// NeuroPLC ¡ª FourierKAN L0-direct configuration [28,16,4]
// L0 (28->16): analytic SIN/COS harmonics + SiLU base (no LUT)
// L1 (16->4): LUT N=16 on [-3.15, 3.15] (100% L0-out coverage)
// Sound bound 0.130 (safety 5.2x) ¡ª verify_fourier_l0direct.py
FUNCTION_BLOCK "NeuroPLC_FourierKAN_L0DIR"
VAR_INPUT
    "feat_1" : REAL;
    "feat_2" : REAL;
    "feat_3" : REAL;
    "feat_4" : REAL;
    "feat_5" : REAL;
    "feat_6" : REAL;
    "feat_7" : REAL;
    "feat_8" : REAL;
    "feat_9" : REAL;
    "feat_10" : REAL;
    "feat_11" : REAL;
    "feat_12" : REAL;
    "feat_13" : REAL;
    "feat_14" : REAL;
    "feat_15" : REAL;
    "feat_16" : REAL;
    "feat_17" : REAL;
    "feat_18" : REAL;
    "feat_19" : REAL;
    "feat_20" : REAL;
    "feat_21" : REAL;
    "feat_22" : REAL;
    "feat_23" : REAL;
    "feat_24" : REAL;
    "feat_25" : REAL;
    "feat_26" : REAL;
    "feat_27" : REAL;
    "feat_28" : REAL;
    "trigger" : BOOL;
END_VAR
VAR_OUTPUT
    "class_1" : REAL;
    "class_2" : REAL;
    "class_3" : REAL;
    "class_4" : REAL;
    "pred_class" : INT;
END_VAR
VAR
    "h1_1" : REAL := 0.0;
    "h1_2" : REAL := 0.0;
    "h1_3" : REAL := 0.0;
    "h1_4" : REAL := 0.0;
    "h1_5" : REAL := 0.0;
    "h1_6" : REAL := 0.0;
    "h1_7" : REAL := 0.0;
    "h1_8" : REAL := 0.0;
    "h1_9" : REAL := 0.0;
    "h1_10" : REAL := 0.0;
    "h1_11" : REAL := 0.0;
    "h1_12" : REAL := 0.0;
    "h1_13" : REAL := 0.0;
    "h1_14" : REAL := 0.0;
    "h1_15" : REAL := 0.0;
    "h1_16" : REAL := 0.0;
    "x" : REAL; "phi" : REAL; "acc" : REAL := 0.0;
    "i" : INT; "j" : INT; "k" : INT;
    "lo" : INT; "hi" : INT; "mid" : INT; "t" : REAL;
END_VAR

BEGIN
    IF NOT "trigger" THEN RETURN; END_IF;

    // === L0 (28->16): analytic FourierKAN ===
    "acc" := 0.0;
    "x" := "feat_1";
    "phi" := "w0b_1_1" * "x" / (1.0 + EXP(-"x"));
    "phi" := "phi" + "w0c_1_1_1" * SIN(1 * 0.4 * "x") + "w0d_1_1_1" * COS(1 * 0.4 * "x");
    "phi" := "phi" + "w0c_1_1_2" * SIN(2 * 0.4 * "x") + "w0d_1_1_2" * COS(2 * 0.4 * "x");
    "phi" := "phi" + "w0c_1_1_3" * SIN(3 * 0.4 * "x") + "w0d_1_1_3" * COS(3 * 0.4 * "x");
    "phi" := "phi" + "w0c_1_1_4" * SIN(4 * 0.4 * "x") + "w0d_1_1_4" * COS(4 * 0.4 * "x");
    "phi" := "phi" + "w0c_1_1_5" * SIN(5 * 0.4 * "x") + "w0d_1_1_5" * COS(5 * 0.4 * "x");
    "phi" := "phi" + "w0c_1_1_6" * SIN(6 * 0.4 * "x") + "w0d_1_1_6" * COS(6 * 0.4 * "x");
    "acc" := "acc" + "phi";
    "x" := "feat_2";
    "phi" := "w0b_1_2" * "x" / (1.0 + EXP(-"x"));
    "phi" := "phi" + "w0c_1_2_1" * SIN(1 * 0.4 * "x") + "w0d_1_2_1" * COS(1 * 0.4 * "x");
    "phi" := "phi" + "w0c_1_2_2" * SIN(2 * 0.4 * "x") + "w0d_1_2_2" * COS(2 * 0.4 * "x");
    "phi" := "phi" + "w0c_1_2_3" * SIN(3 * 0.4 * "x") + "w0d_1_2_3" * COS(3 * 0.4 * "x");
    "phi" := "phi" + "w0c_1_2_4" * SIN(4 * 0.4 * "x") + "w0d_1_2_4" * COS(4 * 0.4 * "x");
    "phi" := "phi" + "w0c_1_2_5" * SIN(5 * 0.4 * "x") + "w0d_1_2_5" * COS(5 * 0.4 * "x");
    "phi" := "phi" + "w0c_1_2_6" * SIN(6 * 0.4 * "x") + "w0d_1_2_6" * COS(6 * 0.4 * "x");
    "acc" := "acc" + "phi";
    "x" := "feat_3";
    "phi" := "w0b_1_3" * "x" / (1.0 + EXP(-"x"));
    "phi" := "phi" + "w0c_1_3_1" * SIN(1 * 0.4 * "x") + "w0d_1_3_1" * COS(1 * 0.4 * "x");
    "phi" := "phi" + "w0c_1_3_2" * SIN(2 * 0.4 * "x") + "w0d_1_3_2" * COS(2 * 0.4 * "x");
    "phi" := "phi" + "w0c_1_3_3" * SIN(3 * 0.4 * "x") + "w0d_1_3_3" * COS(3 * 0.4 * "x");
    "phi" := "phi" + "w0c_1_3_4" * SIN(4 * 0.4 * "x") + "w0d_1_3_4" * COS(4 * 0.4 * "x");
    "phi" := "phi" + "w0c_1_3_5" * SIN(5 * 0.4 * "x") + "w0d_1_3_5" * COS(5 * 0.4 * "x");
    "phi" := "phi" + "w0c_1_3_6" * SIN(6 * 0.4 * "x") + "w0d_1_3_6" * COS(6 * 0.4 * "x");
    "acc" := "acc" + "phi";
    "x" := "feat_4";
    "phi" := "w0b_1_4" * "x" / (1.0 + EXP(-"x"));
    "phi" := "phi" + "w0c_1_4_1" * SIN(1 * 0.4 * "x") + "w0d_1_4_1" * COS(1 * 0.4 * "x");
    "phi" := "phi" + "w0c_1_4_2" * SIN(2 * 0.4 * "x") + "w0d_1_4_2" * COS(2 * 0.4 * "x");
    "phi" := "phi" + "w0c_1_4_3" * SIN(3 * 0.4 * "x") + "w0d_1_4_3" * COS(3 * 0.4 * "x");
    "phi" := "phi" + "w0c_1_4_4" * SIN(4 * 0.4 * "x") + "w0d_1_4_4" * COS(4 * 0.4 * "x");
    "phi" := "phi" + "w0c_1_4_5" * SIN(5 * 0.4 * "x") + "w0d_1_4_5" * COS(5 * 0.4 * "x");
    "phi" := "phi" + "w0c_1_4_6" * SIN(6 * 0.4 * "x") + "w0d_1_4_6" * COS(6 * 0.4 * "x");
    "acc" := "acc" + "phi";
    "x" := "feat_5";
    "phi" := "w0b_1_5" * "x" / (1.0 + EXP(-"x"));
    "phi" := "phi" + "w0c_1_5_1" * SIN(1 * 0.4 * "x") + "w0d_1_5_1" * COS(1 * 0.4 * "x");
    "phi" := "phi" + "w0c_1_5_2" * SIN(2 * 0.4 * "x") + "w0d_1_5_2" * COS(2 * 0.4 * "x");
    "phi" := "phi" + "w0c_1_5_3" * SIN(3 * 0.4 * "x") + "w0d_1_5_3" * COS(3 * 0.4 * "x");
    "phi" := "phi" + "w0c_1_5_4" * SIN(4 * 0.4 * "x") + "w0d_1_5_4" * COS(4 * 0.4 * "x");
    "phi" := "phi" + "w0c_1_5_5" * SIN(5 * 0.4 * "x") + "w0d_1_5_5" * COS(5 * 0.4 * "x");
    "phi" := "phi" + "w0c_1_5_6" * SIN(6 * 0.4 * "x") + "w0d_1_5_6" * COS(6 * 0.4 * "x");
    "acc" := "acc" + "phi";
    "x" := "feat_6";
    "phi" := "w0b_1_6" * "x" / (1.0 + EXP(-"x"));
    "phi" := "phi" + "w0c_1_6_1" * SIN(1 * 0.4 * "x") + "w0d_1_6_1" * COS(1 * 0.4 * "x");
    "phi" := "phi" + "w0c_1_6_2" * SIN(2 * 0.4 * "x") + "w0d_1_6_2" * COS(2 * 0.4 * "x");
    "phi" := "phi" + "w0c_1_6_3" * SIN(3 * 0.4 * "x") + "w0d_1_6_3" * COS(3 * 0.4 * "x");
    "phi" := "phi" + "w0c_1_6_4" * SIN(4 * 0.4 * "x") + "w0d_1_6_4" * COS(4 * 0.4 * "x");
    "phi" := "phi" + "w0c_1_6_5" * SIN(5 * 0.4 * "x") + "w0d_1_6_5" * COS(5 * 0.4 * "x");
    "phi" := "phi" + "w0c_1_6_6" * SIN(6 * 0.4 * "x") + "w0d_1_6_6" * COS(6 * 0.4 * "x");
    "acc" := "acc" + "phi";
    "x" := "feat_7";
    "phi" := "w0b_1_7" * "x" / (1.0 + EXP(-"x"));
    "phi" := "phi" + "w0c_1_7_1" * SIN(1 * 0.4 * "x") + "w0d_1_7_1" * COS(1 * 0.4 * "x");
    "phi" := "phi" + "w0c_1_7_2" * SIN(2 * 0.4 * "x") + "w0d_1_7_2" * COS(2 * 0.4 * "x");
    "phi" := "phi" + "w0c_1_7_3" * SIN(3 * 0.4 * "x") + "w0d_1_7_3" * COS(3 * 0.4 * "x");
    "phi" := "phi" + "w0c_1_7_4" * SIN(4 * 0.4 * "x") + "w0d_1_7_4" * COS(4 * 0.4 * "x");
    "phi" := "phi" + "w0c_1_7_5" * SIN(5 * 0.4 * "x") + "w0d_1_7_5" * COS(5 * 0.4 * "x");
    "phi" := "phi" + "w0c_1_7_6" * SIN(6 * 0.4 * "x") + "w0d_1_7_6" * COS(6 * 0.4 * "x");
    "acc" := "acc" + "phi";
    "x" := "feat_8";
    "phi" := "w0b_1_8" * "x" / (1.0 + EXP(-"x"));
    "phi" := "phi" + "w0c_1_8_1" * SIN(1 * 0.4 * "x") + "w0d_1_8_1" * COS(1 * 0.4 * "x");
    "phi" := "phi" + "w0c_1_8_2" * SIN(2 * 0.4 * "x") + "w0d_1_8_2" * COS(2 * 0.4 * "x");
    "phi" := "phi" + "w0c_1_8_3" * SIN(3 * 0.4 * "x") + "w0d_1_8_3" * COS(3 * 0.4 * "x");
    "phi" := "phi" + "w0c_1_8_4" * SIN(4 * 0.4 * "x") + "w0d_1_8_4" * COS(4 * 0.4 * "x");
    "phi" := "phi" + "w0c_1_8_5" * SIN(5 * 0.4 * "x") + "w0d_1_8_5" * COS(5 * 0.4 * "x");
    "phi" := "phi" + "w0c_1_8_6" * SIN(6 * 0.4 * "x") + "w0d_1_8_6" * COS(6 * 0.4 * "x");
    "acc" := "acc" + "phi";
    "x" := "feat_9";
    "phi" := "w0b_1_9" * "x" / (1.0 + EXP(-"x"));
    "phi" := "phi" + "w0c_1_9_1" * SIN(1 * 0.4 * "x") + "w0d_1_9_1" * COS(1 * 0.4 * "x");
    "phi" := "phi" + "w0c_1_9_2" * SIN(2 * 0.4 * "x") + "w0d_1_9_2" * COS(2 * 0.4 * "x");
    "phi" := "phi" + "w0c_1_9_3" * SIN(3 * 0.4 * "x") + "w0d_1_9_3" * COS(3 * 0.4 * "x");
    "phi" := "phi" + "w0c_1_9_4" * SIN(4 * 0.4 * "x") + "w0d_1_9_4" * COS(4 * 0.4 * "x");
    "phi" := "phi" + "w0c_1_9_5" * SIN(5 * 0.4 * "x") + "w0d_1_9_5" * COS(5 * 0.4 * "x");
    "phi" := "phi" + "w0c_1_9_6" * SIN(6 * 0.4 * "x") + "w0d_1_9_6" * COS(6 * 0.4 * "x");
    "acc" := "acc" + "phi";
    "x" := "feat_10";
    "phi" := "w0b_1_10" * "x" / (1.0 + EXP(-"x"));
    "phi" := "phi" + "w0c_1_10_1" * SIN(1 * 0.4 * "x") + "w0d_1_10_1" * COS(1 * 0.4 * "x");
    "phi" := "phi" + "w0c_1_10_2" * SIN(2 * 0.4 * "x") + "w0d_1_10_2" * COS(2 * 0.4 * "x");
    "phi" := "phi" + "w0c_1_10_3" * SIN(3 * 0.4 * "x") + "w0d_1_10_3" * COS(3 * 0.4 * "x");
    "phi" := "phi" + "w0c_1_10_4" * SIN(4 * 0.4 * "x") + "w0d_1_10_4" * COS(4 * 0.4 * "x");
    "phi" := "phi" + "w0c_1_10_5" * SIN(5 * 0.4 * "x") + "w0d_1_10_5" * COS(5 * 0.4 * "x");
    "phi" := "phi" + "w0c_1_10_6" * SIN(6 * 0.4 * "x") + "w0d_1_10_6" * COS(6 * 0.4 * "x");
    "acc" := "acc" + "phi";
    "x" := "feat_11";
    "phi" := "w0b_1_11" * "x" / (1.0 + EXP(-"x"));
    "phi" := "phi" + "w0c_1_11_1" * SIN(1 * 0.4 * "x") + "w0d_1_11_1" * COS(1 * 0.4 * "x");
    "phi" := "phi" + "w0c_1_11_2" * SIN(2 * 0.4 * "x") + "w0d_1_11_2" * COS(2 * 0.4 * "x");
    "phi" := "phi" + "w0c_1_11_3" * SIN(3 * 0.4 * "x") + "w0d_1_11_3" * COS(3 * 0.4 * "x");
    "phi" := "phi" + "w0c_1_11_4" * SIN(4 * 0.4 * "x") + "w0d_1_11_4" * COS(4 * 0.4 * "x");
    "phi" := "phi" + "w0c_1_11_5" * SIN(5 * 0.4 * "x") + "w0d_1_11_5" * COS(5 * 0.4 * "x");
    "phi" := "phi" + "w0c_1_11_6" * SIN(6 * 0.4 * "x") + "w0d_1_11_6" * COS(6 * 0.4 * "x");
    "acc" := "acc" + "phi";
    "x" := "feat_12";
    "phi" := "w0b_1_12" * "x" / (1.0 + EXP(-"x"));
    "phi" := "phi" + "w0c_1_12_1" * SIN(1 * 0.4 * "x") + "w0d_1_12_1" * COS(1 * 0.4 * "x");
    "phi" := "phi" + "w0c_1_12_2" * SIN(2 * 0.4 * "x") + "w0d_1_12_2" * COS(2 * 0.4 * "x");
    "phi" := "phi" + "w0c_1_12_3" * SIN(3 * 0.4 * "x") + "w0d_1_12_3" * COS(3 * 0.4 * "x");
    "phi" := "phi" + "w0c_1_12_4" * SIN(4 * 0.4 * "x") + "w0d_1_12_4" * COS(4 * 0.4 * "x");
    "phi" := "phi" + "w0c_1_12_5" * SIN(5 * 0.4 * "x") + "w0d_1_12_5" * COS(5 * 0.4 * "x");
    "phi" := "phi" + "w0c_1_12_6" * SIN(6 * 0.4 * "x") + "w0d_1_12_6" * COS(6 * 0.4 * "x");
    "acc" := "acc" + "phi";
    "x" := "feat_13";
    "phi" := "w0b_1_13" * "x" / (1.0 + EXP(-"x"));
    "phi" := "phi" + "w0c_1_13_1" * SIN(1 * 0.4 * "x") + "w0d_1_13_1" * COS(1 * 0.4 * "x");
    "phi" := "phi" + "w0c_1_13_2" * SIN(2 * 0.4 * "x") + "w0d_1_13_2" * COS(2 * 0.4 * "x");
    "phi" := "phi" + "w0c_1_13_3" * SIN(3 * 0.4 * "x") + "w0d_1_13_3" * COS(3 * 0.4 * "x");
    "phi" := "phi" + "w0c_1_13_4" * SIN(4 * 0.4 * "x") + "w0d_1_13_4" * COS(4 * 0.4 * "x");
    "phi" := "phi" + "w0c_1_13_5" * SIN(5 * 0.4 * "x") + "w0d_1_13_5" * COS(5 * 0.4 * "x");
    "phi" := "phi" + "w0c_1_13_6" * SIN(6 * 0.4 * "x") + "w0d_1_13_6" * COS(6 * 0.4 * "x");
    "acc" := "acc" + "phi";
    "x" := "feat_14";
    "phi" := "w0b_1_14" * "x" / (1.0 + EXP(-"x"));
    "phi" := "phi" + "w0c_1_14_1" * SIN(1 * 0.4 * "x") + "w0d_1_14_1" * COS(1 * 0.4 * "x");
    "phi" := "phi" + "w0c_1_14_2" * SIN(2 * 0.4 * "x") + "w0d_1_14_2" * COS(2 * 0.4 * "x");
    "phi" := "phi" + "w0c_1_14_3" * SIN(3 * 0.4 * "x") + "w0d_1_14_3" * COS(3 * 0.4 * "x");
    "phi" := "phi" + "w0c_1_14_4" * SIN(4 * 0.4 * "x") + "w0d_1_14_4" * COS(4 * 0.4 * "x");
    "phi" := "phi" + "w0c_1_14_5" * SIN(5 * 0.4 * "x") + "w0d_1_14_5" * COS(5 * 0.4 * "x");
    "phi" := "phi" + "w0c_1_14_6" * SIN(6 * 0.4 * "x") + "w0d_1_14_6" * COS(6 * 0.4 * "x");
    "acc" := "acc" + "phi";
    "x" := "feat_15";
    "phi" := "w0b_1_15" * "x" / (1.0 + EXP(-"x"));
    "phi" := "phi" + "w0c_1_15_1" * SIN(1 * 0.4 * "x") + "w0d_1_15_1" * COS(1 * 0.4 * "x");
    "phi" := "phi" + "w0c_1_15_2" * SIN(2 * 0.4 * "x") + "w0d_1_15_2" * COS(2 * 0.4 * "x");
    "phi" := "phi" + "w0c_1_15_3" * SIN(3 * 0.4 * "x") + "w0d_1_15_3" * COS(3 * 0.4 * "x");
    "phi" := "phi" + "w0c_1_15_4" * SIN(4 * 0.4 * "x") + "w0d_1_15_4" * COS(4 * 0.4 * "x");
    "phi" := "phi" + "w0c_1_15_5" * SIN(5 * 0.4 * "x") + "w0d_1_15_5" * COS(5 * 0.4 * "x");
    "phi" := "phi" + "w0c_1_15_6" * SIN(6 * 0.4 * "x") + "w0d_1_15_6" * COS(6 * 0.4 * "x");
    "acc" := "acc" + "phi";
    "x" := "feat_16";
    "phi" := "w0b_1_16" * "x" / (1.0 + EXP(-"x"));
    "phi" := "phi" + "w0c_1_16_1" * SIN(1 * 0.4 * "x") + "w0d_1_16_1" * COS(1 * 0.4 * "x");
    "phi" := "phi" + "w0c_1_16_2" * SIN(2 * 0.4 * "x") + "w0d_1_16_2" * COS(2 * 0.4 * "x");
    "phi" := "phi" + "w0c_1_16_3" * SIN(3 * 0.4 * "x") + "w0d_1_16_3" * COS(3 * 0.4 * "x");
    "phi" := "phi" + "w0c_1_16_4" * SIN(4 * 0.4 * "x") + "w0d_1_16_4" * COS(4 * 0.4 * "x");
    "phi" := "phi" + "w0c_1_16_5" * SIN(5 * 0.4 * "x") + "w0d_1_16_5" * COS(5 * 0.4 * "x");
    "phi" := "phi" + "w0c_1_16_6" * SIN(6 * 0.4 * "x") + "w0d_1_16_6" * COS(6 * 0.4 * "x");
    "acc" := "acc" + "phi";
    "x" := "feat_17";
    "phi" := "w0b_1_17" * "x" / (1.0 + EXP(-"x"));
    "phi" := "phi" + "w0c_1_17_1" * SIN(1 * 0.4 * "x") + "w0d_1_17_1" * COS(1 * 0.4 * "x");
    "phi" := "phi" + "w0c_1_17_2" * SIN(2 * 0.4 * "x") + "w0d_1_17_2" * COS(2 * 0.4 * "x");
    "phi" := "phi" + "w0c_1_17_3" * SIN(3 * 0.4 * "x") + "w0d_1_17_3" * COS(3 * 0.4 * "x");
    "phi" := "phi" + "w0c_1_17_4" * SIN(4 * 0.4 * "x") + "w0d_1_17_4" * COS(4 * 0.4 * "x");
    "phi" := "phi" + "w0c_1_17_5" * SIN(5 * 0.4 * "x") + "w0d_1_17_5" * COS(5 * 0.4 * "x");
    "phi" := "phi" + "w0c_1_17_6" * SIN(6 * 0.4 * "x") + "w0d_1_17_6" * COS(6 * 0.4 * "x");
    "acc" := "acc" + "phi";
    "x" := "feat_18";
    "phi" := "w0b_1_18" * "x" / (1.0 + EXP(-"x"));
    "phi" := "phi" + "w0c_1_18_1" * SIN(1 * 0.4 * "x") + "w0d_1_18_1" * COS(1 * 0.4 * "x");
    "phi" := "phi" + "w0c_1_18_2" * SIN(2 * 0.4 * "x") + "w0d_1_18_2" * COS(2 * 0.4 * "x");
    "phi" := "phi" + "w0c_1_18_3" * SIN(3 * 0.4 * "x") + "w0d_1_18_3" * COS(3 * 0.4 * "x");
    "phi" := "phi" + "w0c_1_18_4" * SIN(4 * 0.4 * "x") + "w0d_1_18_4" * COS(4 * 0.4 * "x");
    "phi" := "phi" + "w0c_1_18_5" * SIN(5 * 0.4 * "x") + "w0d_1_18_5" * COS(5 * 0.4 * "x");
    "phi" := "phi" + "w0c_1_18_6" * SIN(6 * 0.4 * "x") + "w0d_1_18_6" * COS(6 * 0.4 * "x");
    "acc" := "acc" + "phi";
    "x" := "feat_19";
    "phi" := "w0b_1_19" * "x" / (1.0 + EXP(-"x"));
    "phi" := "phi" + "w0c_1_19_1" * SIN(1 * 0.4 * "x") + "w0d_1_19_1" * COS(1 * 0.4 * "x");
    "phi" := "phi" + "w0c_1_19_2" * SIN(2 * 0.4 * "x") + "w0d_1_19_2" * COS(2 * 0.4 * "x");
    "phi" := "phi" + "w0c_1_19_3" * SIN(3 * 0.4 * "x") + "w0d_1_19_3" * COS(3 * 0.4 * "x");
    "phi" := "phi" + "w0c_1_19_4" * SIN(4 * 0.4 * "x") + "w0d_1_19_4" * COS(4 * 0.4 * "x");
    "phi" := "phi" + "w0c_1_19_5" * SIN(5 * 0.4 * "x") + "w0d_1_19_5" * COS(5 * 0.4 * "x");
    "phi" := "phi" + "w0c_1_19_6" * SIN(6 * 0.4 * "x") + "w0d_1_19_6" * COS(6 * 0.4 * "x");
    "acc" := "acc" + "phi";
    "x" := "feat_20";
    "phi" := "w0b_1_20" * "x" / (1.0 + EXP(-"x"));
    "phi" := "phi" + "w0c_1_20_1" * SIN(1 * 0.4 * "x") + "w0d_1_20_1" * COS(1 * 0.4 * "x");
    "phi" := "phi" + "w0c_1_20_2" * SIN(2 * 0.4 * "x") + "w0d_1_20_2" * COS(2 * 0.4 * "x");
    "phi" := "phi" + "w0c_1_20_3" * SIN(3 * 0.4 * "x") + "w0d_1_20_3" * COS(3 * 0.4 * "x");
    "phi" := "phi" + "w0c_1_20_4" * SIN(4 * 0.4 * "x") + "w0d_1_20_4" * COS(4 * 0.4 * "x");
    "phi" := "phi" + "w0c_1_20_5" * SIN(5 * 0.4 * "x") + "w0d_1_20_5" * COS(5 * 0.4 * "x");
    "phi" := "phi" + "w0c_1_20_6" * SIN(6 * 0.4 * "x") + "w0d_1_20_6" * COS(6 * 0.4 * "x");
    "acc" := "acc" + "phi";
    "x" := "feat_21";
    "phi" := "w0b_1_21" * "x" / (1.0 + EXP(-"x"));
    "phi" := "phi" + "w0c_1_21_1" * SIN(1 * 0.4 * "x") + "w0d_1_21_1" * COS(1 * 0.4 * "x");
    "phi" := "phi" + "w0c_1_21_2" * SIN(2 * 0.4 * "x") + "w0d_1_21_2" * COS(2 * 0.4 * "x");
    "phi" := "phi" + "w0c_1_21_3" * SIN(3 * 0.4 * "x") + "w0d_1_21_3" * COS(3 * 0.4 * "x");
    "phi" := "phi" + "w0c_1_21_4" * SIN(4 * 0.4 * "x") + "w0d_1_21_4" * COS(4 * 0.4 * "x");
    "phi" := "phi" + "w0c_1_21_5" * SIN(5 * 0.4 * "x") + "w0d_1_21_5" * COS(5 * 0.4 * "x");
    "phi" := "phi" + "w0c_1_21_6" * SIN(6 * 0.4 * "x") + "w0d_1_21_6" * COS(6 * 0.4 * "x");
    "acc" := "acc" + "phi";
    "x" := "feat_22";
    "phi" := "w0b_1_22" * "x" / (1.0 + EXP(-"x"));
    "phi" := "phi" + "w0c_1_22_1" * SIN(1 * 0.4 * "x") + "w0d_1_22_1" * COS(1 * 0.4 * "x");
    "phi" := "phi" + "w0c_1_22_2" * SIN(2 * 0.4 * "x") + "w0d_1_22_2" * COS(2 * 0.4 * "x");
    "phi" := "phi" + "w0c_1_22_3" * SIN(3 * 0.4 * "x") + "w0d_1_22_3" * COS(3 * 0.4 * "x");
    "phi" := "phi" + "w0c_1_22_4" * SIN(4 * 0.4 * "x") + "w0d_1_22_4" * COS(4 * 0.4 * "x");
    "phi" := "phi" + "w0c_1_22_5" * SIN(5 * 0.4 * "x") + "w0d_1_22_5" * COS(5 * 0.4 * "x");
    "phi" := "phi" + "w0c_1_22_6" * SIN(6 * 0.4 * "x") + "w0d_1_22_6" * COS(6 * 0.4 * "x");
    "acc" := "acc" + "phi";
    "x" := "feat_23";
    "phi" := "w0b_1_23" * "x" / (1.0 + EXP(-"x"));
    "phi" := "phi" + "w0c_1_23_1" * SIN(1 * 0.4 * "x") + "w0d_1_23_1" * COS(1 * 0.4 * "x");
    "phi" := "phi" + "w0c_1_23_2" * SIN(2 * 0.4 * "x") + "w0d_1_23_2" * COS(2 * 0.4 * "x");
    "phi" := "phi" + "w0c_1_23_3" * SIN(3 * 0.4 * "x") + "w0d_1_23_3" * COS(3 * 0.4 * "x");
    "phi" := "phi" + "w0c_1_23_4" * SIN(4 * 0.4 * "x") + "w0d_1_23_4" * COS(4 * 0.4 * "x");
    "phi" := "phi" + "w0c_1_23_5" * SIN(5 * 0.4 * "x") + "w0d_1_23_5" * COS(5 * 0.4 * "x");
    "phi" := "phi" + "w0c_1_23_6" * SIN(6 * 0.4 * "x") + "w0d_1_23_6" * COS(6 * 0.4 * "x");
    "acc" := "acc" + "phi";
    "x" := "feat_24";
    "phi" := "w0b_1_24" * "x" / (1.0 + EXP(-"x"));
    "phi" := "phi" + "w0c_1_24_1" * SIN(1 * 0.4 * "x") + "w0d_1_24_1" * COS(1 * 0.4 * "x");
    "phi" := "phi" + "w0c_1_24_2" * SIN(2 * 0.4 * "x") + "w0d_1_24_2" * COS(2 * 0.4 * "x");
    "phi" := "phi" + "w0c_1_24_3" * SIN(3 * 0.4 * "x") + "w0d_1_24_3" * COS(3 * 0.4 * "x");
    "phi" := "phi" + "w0c_1_24_4" * SIN(4 * 0.4 * "x") + "w0d_1_24_4" * COS(4 * 0.4 * "x");
    "phi" := "phi" + "w0c_1_24_5" * SIN(5 * 0.4 * "x") + "w0d_1_24_5" * COS(5 * 0.4 * "x");
    "phi" := "phi" + "w0c_1_24_6" * SIN(6 * 0.4 * "x") + "w0d_1_24_6" * COS(6 * 0.4 * "x");
    "acc" := "acc" + "phi";
    "x" := "feat_25";
    "phi" := "w0b_1_25" * "x" / (1.0 + EXP(-"x"));
    "phi" := "phi" + "w0c_1_25_1" * SIN(1 * 0.4 * "x") + "w0d_1_25_1" * COS(1 * 0.4 * "x");
    "phi" := "phi" + "w0c_1_25_2" * SIN(2 * 0.4 * "x") + "w0d_1_25_2" * COS(2 * 0.4 * "x");
    "phi" := "phi" + "w0c_1_25_3" * SIN(3 * 0.4 * "x") + "w0d_1_25_3" * COS(3 * 0.4 * "x");
    "phi" := "phi" + "w0c_1_25_4" * SIN(4 * 0.4 * "x") + "w0d_1_25_4" * COS(4 * 0.4 * "x");
    "phi" := "phi" + "w0c_1_25_5" * SIN(5 * 0.4 * "x") + "w0d_1_25_5" * COS(5 * 0.4 * "x");
    "phi" := "phi" + "w0c_1_25_6" * SIN(6 * 0.4 * "x") + "w0d_1_25_6" * COS(6 * 0.4 * "x");
    "acc" := "acc" + "phi";
    "x" := "feat_26";
    "phi" := "w0b_1_26" * "x" / (1.0 + EXP(-"x"));
    "phi" := "phi" + "w0c_1_26_1" * SIN(1 * 0.4 * "x") + "w0d_1_26_1" * COS(1 * 0.4 * "x");
    "phi" := "phi" + "w0c_1_26_2" * SIN(2 * 0.4 * "x") + "w0d_1_26_2" * COS(2 * 0.4 * "x");
    "phi" := "phi" + "w0c_1_26_3" * SIN(3 * 0.4 * "x") + "w0d_1_26_3" * COS(3 * 0.4 * "x");
    "phi" := "phi" + "w0c_1_26_4" * SIN(4 * 0.4 * "x") + "w0d_1_26_4" * COS(4 * 0.4 * "x");
    "phi" := "phi" + "w0c_1_26_5" * SIN(5 * 0.4 * "x") + "w0d_1_26_5" * COS(5 * 0.4 * "x");
    "phi" := "phi" + "w0c_1_26_6" * SIN(6 * 0.4 * "x") + "w0d_1_26_6" * COS(6 * 0.4 * "x");
    "acc" := "acc" + "phi";
    "x" := "feat_27";
    "phi" := "w0b_1_27" * "x" / (1.0 + EXP(-"x"));
    "phi" := "phi" + "w0c_1_27_1" * SIN(1 * 0.4 * "x") + "w0d_1_27_1" * COS(1 * 0.4 * "x");
    "phi" := "phi" + "w0c_1_27_2" * SIN(2 * 0.4 * "x") + "w0d_1_27_2" * COS(2 * 0.4 * "x");
    "phi" := "phi" + "w0c_1_27_3" * SIN(3 * 0.4 * "x") + "w0d_1_27_3" * COS(3 * 0.4 * "x");
    "phi" := "phi" + "w0c_1_27_4" * SIN(4 * 0.4 * "x") + "w0d_1_27_4" * COS(4 * 0.4 * "x");
    "phi" := "phi" + "w0c_1_27_5" * SIN(5 * 0.4 * "x") + "w0d_1_27_5" * COS(5 * 0.4 * "x");
    "phi" := "phi" + "w0c_1_27_6" * SIN(6 * 0.4 * "x") + "w0d_1_27_6" * COS(6 * 0.4 * "x");
    "acc" := "acc" + "phi";
    "x" := "feat_28";
    "phi" := "w0b_1_28" * "x" / (1.0 + EXP(-"x"));
    "phi" := "phi" + "w0c_1_28_1" * SIN(1 * 0.4 * "x") + "w0d_1_28_1" * COS(1 * 0.4 * "x");
    "phi" := "phi" + "w0c_1_28_2" * SIN(2 * 0.4 * "x") + "w0d_1_28_2" * COS(2 * 0.4 * "x");
    "phi" := "phi" + "w0c_1_28_3" * SIN(3 * 0.4 * "x") + "w0d_1_28_3" * COS(3 * 0.4 * "x");
    "phi" := "phi" + "w0c_1_28_4" * SIN(4 * 0.4 * "x") + "w0d_1_28_4" * COS(4 * 0.4 * "x");
    "phi" := "phi" + "w0c_1_28_5" * SIN(5 * 0.4 * "x") + "w0d_1_28_5" * COS(5 * 0.4 * "x");
    "phi" := "phi" + "w0c_1_28_6" * SIN(6 * 0.4 * "x") + "w0d_1_28_6" * COS(6 * 0.4 * "x");
    "acc" := "acc" + "phi";
    "h1_1" := "acc" + "b0_1";
    "acc" := 0.0;
    "x" := "feat_1";
    "phi" := "w0b_2_1" * "x" / (1.0 + EXP(-"x"));
    "phi" := "phi" + "w0c_2_1_1" * SIN(1 * 0.4 * "x") + "w0d_2_1_1" * COS(1 * 0.4 * "x");
    "phi" := "phi" + "w0c_2_1_2" * SIN(2 * 0.4 * "x") + "w0d_2_1_2" * COS(2 * 0.4 * "x");
    "phi" := "phi" + "w0c_2_1_3" * SIN(3 * 0.4 * "x") + "w0d_2_1_3" * COS(3 * 0.4 * "x");
    "phi" := "phi" + "w0c_2_1_4" * SIN(4 * 0.4 * "x") + "w0d_2_1_4" * COS(4 * 0.4 * "x");
    "phi" := "phi" + "w0c_2_1_5" * SIN(5 * 0.4 * "x") + "w0d_2_1_5" * COS(5 * 0.4 * "x");
    "phi" := "phi" + "w0c_2_1_6" * SIN(6 * 0.4 * "x") + "w0d_2_1_6" * COS(6 * 0.4 * "x");
    "acc" := "acc" + "phi";
    "x" := "feat_2";
    "phi" := "w0b_2_2" * "x" / (1.0 + EXP(-"x"));
    "phi" := "phi" + "w0c_2_2_1" * SIN(1 * 0.4 * "x") + "w0d_2_2_1" * COS(1 * 0.4 * "x");
    "phi" := "phi" + "w0c_2_2_2" * SIN(2 * 0.4 * "x") + "w0d_2_2_2" * COS(2 * 0.4 * "x");
    "phi" := "phi" + "w0c_2_2_3" * SIN(3 * 0.4 * "x") + "w0d_2_2_3" * COS(3 * 0.4 * "x");
    "phi" := "phi" + "w0c_2_2_4" * SIN(4 * 0.4 * "x") + "w0d_2_2_4" * COS(4 * 0.4 * "x");
    "phi" := "phi" + "w0c_2_2_5" * SIN(5 * 0.4 * "x") + "w0d_2_2_5" * COS(5 * 0.4 * "x");
    "phi" := "phi" + "w0c_2_2_6" * SIN(6 * 0.4 * "x") + "w0d_2_2_6" * COS(6 * 0.4 * "x");
    "acc" := "acc" + "phi";
    "x" := "feat_3";
    "phi" := "w0b_2_3" * "x" / (1.0 + EXP(-"x"));
    "phi" := "phi" + "w0c_2_3_1" * SIN(1 * 0.4 * "x") + "w0d_2_3_1" * COS(1 * 0.4 * "x");
    "phi" := "phi" + "w0c_2_3_2" * SIN(2 * 0.4 * "x") + "w0d_2_3_2" * COS(2 * 0.4 * "x");
    "phi" := "phi" + "w0c_2_3_3" * SIN(3 * 0.4 * "x") + "w0d_2_3_3" * COS(3 * 0.4 * "x");
    "phi" := "phi" + "w0c_2_3_4" * SIN(4 * 0.4 * "x") + "w0d_2_3_4" * COS(4 * 0.4 * "x");
    "phi" := "phi" + "w0c_2_3_5" * SIN(5 * 0.4 * "x") + "w0d_2_3_5" * COS(5 * 0.4 * "x");
    "phi" := "phi" + "w0c_2_3_6" * SIN(6 * 0.4 * "x") + "w0d_2_3_6" * COS(6 * 0.4 * "x");
    "acc" := "acc" + "phi";
    "x" := "feat_4";
    "phi" := "w0b_2_4" * "x" / (1.0 + EXP(-"x"));
    "phi" := "phi" + "w0c_2_4_1" * SIN(1 * 0.4 * "x") + "w0d_2_4_1" * COS(1 * 0.4 * "x");
    "phi" := "phi" + "w0c_2_4_2" * SIN(2 * 0.4 * "x") + "w0d_2_4_2" * COS(2 * 0.4 * "x");
    "phi" := "phi" + "w0c_2_4_3" * SIN(3 * 0.4 * "x") + "w0d_2_4_3" * COS(3 * 0.4 * "x");
    "phi" := "phi" + "w0c_2_4_4" * SIN(4 * 0.4 * "x") + "w0d_2_4_4" * COS(4 * 0.4 * "x");
    "phi" := "phi" + "w0c_2_4_5" * SIN(5 * 0.4 * "x") + "w0d_2_4_5" * COS(5 * 0.4 * "x");
    "phi" := "phi" + "w0c_2_4_6" * SIN(6 * 0.4 * "x") + "w0d_2_4_6" * COS(6 * 0.4 * "x");
    "acc" := "acc" + "phi";
    "x" := "feat_5";
    "phi" := "w0b_2_5" * "x" / (1.0 + EXP(-"x"));
    "phi" := "phi" + "w0c_2_5_1" * SIN(1 * 0.4 * "x") + "w0d_2_5_1" * COS(1 * 0.4 * "x");
    "phi" := "phi" + "w0c_2_5_2" * SIN(2 * 0.4 * "x") + "w0d_2_5_2" * COS(2 * 0.4 * "x");
    "phi" := "phi" + "w0c_2_5_3" * SIN(3 * 0.4 * "x") + "w0d_2_5_3" * COS(3 * 0.4 * "x");
    "phi" := "phi" + "w0c_2_5_4" * SIN(4 * 0.4 * "x") + "w0d_2_5_4" * COS(4 * 0.4 * "x");
    "phi" := "phi" + "w0c_2_5_5" * SIN(5 * 0.4 * "x") + "w0d_2_5_5" * COS(5 * 0.4 * "x");
    "phi" := "phi" + "w0c_2_5_6" * SIN(6 * 0.4 * "x") + "w0d_2_5_6" * COS(6 * 0.4 * "x");
    "acc" := "acc" + "phi";
    "x" := "feat_6";
    "phi" := "w0b_2_6" * "x" / (1.0 + EXP(-"x"));
    "phi" := "phi" + "w0c_2_6_1" * SIN(1 * 0.4 * "x") + "w0d_2_6_1" * COS(1 * 0.4 * "x");
    "phi" := "phi" + "w0c_2_6_2" * SIN(2 * 0.4 * "x") + "w0d_2_6_2" * COS(2 * 0.4 * "x");
    "phi" := "phi" + "w0c_2_6_3" * SIN(3 * 0.4 * "x") + "w0d_2_6_3" * COS(3 * 0.4 * "x");
    "phi" := "phi" + "w0c_2_6_4" * SIN(4 * 0.4 * "x") + "w0d_2_6_4" * COS(4 * 0.4 * "x");
    "phi" := "phi" + "w0c_2_6_5" * SIN(5 * 0.4 * "x") + "w0d_2_6_5" * COS(5 * 0.4 * "x");
    "phi" := "phi" + "w0c_2_6_6" * SIN(6 * 0.4 * "x") + "w0d_2_6_6" * COS(6 * 0.4 * "x");
    "acc" := "acc" + "phi";
    "x" := "feat_7";
    "phi" := "w0b_2_7" * "x" / (1.0 + EXP(-"x"));
    "phi" := "phi" + "w0c_2_7_1" * SIN(1 * 0.4 * "x") + "w0d_2_7_1" * COS(1 * 0.4 * "x");
    "phi" := "phi" + "w0c_2_7_2" * SIN(2 * 0.4 * "x") + "w0d_2_7_2" * COS(2 * 0.4 * "x");
    "phi" := "phi" + "w0c_2_7_3" * SIN(3 * 0.4 * "x") + "w0d_2_7_3" * COS(3 * 0.4 * "x");
    "phi" := "phi" + "w0c_2_7_4" * SIN(4 * 0.4 * "x") + "w0d_2_7_4" * COS(4 * 0.4 * "x");
    "phi" := "phi" + "w0c_2_7_5" * SIN(5 * 0.4 * "x") + "w0d_2_7_5" * COS(5 * 0.4 * "x");
    "phi" := "phi" + "w0c_2_7_6" * SIN(6 * 0.4 * "x") + "w0d_2_7_6" * COS(6 * 0.4 * "x");
    "acc" := "acc" + "phi";
    "x" := "feat_8";
    "phi" := "w0b_2_8" * "x" / (1.0 + EXP(-"x"));
    "phi" := "phi" + "w0c_2_8_1" * SIN(1 * 0.4 * "x") + "w0d_2_8_1" * COS(1 * 0.4 * "x");
    "phi" := "phi" + "w0c_2_8_2" * SIN(2 * 0.4 * "x") + "w0d_2_8_2" * COS(2 * 0.4 * "x");
    "phi" := "phi" + "w0c_2_8_3" * SIN(3 * 0.4 * "x") + "w0d_2_8_3" * COS(3 * 0.4 * "x");
    "phi" := "phi" + "w0c_2_8_4" * SIN(4 * 0.4 * "x") + "w0d_2_8_4" * COS(4 * 0.4 * "x");
    "phi" := "phi" + "w0c_2_8_5" * SIN(5 * 0.4 * "x") + "w0d_2_8_5" * COS(5 * 0.4 * "x");
    "phi" := "phi" + "w0c_2_8_6" * SIN(6 * 0.4 * "x") + "w0d_2_8_6" * COS(6 * 0.4 * "x");
    "acc" := "acc" + "phi";
    "x" := "feat_9";
    "phi" := "w0b_2_9" * "x" / (1.0 + EXP(-"x"));
    "phi" := "phi" + "w0c_2_9_1" * SIN(1 * 0.4 * "x") + "w0d_2_9_1" * COS(1 * 0.4 * "x");
    "phi" := "phi" + "w0c_2_9_2" * SIN(2 * 0.4 * "x") + "w0d_2_9_2" * COS(2 * 0.4 * "x");
    "phi" := "phi" + "w0c_2_9_3" * SIN(3 * 0.4 * "x") + "w0d_2_9_3" * COS(3 * 0.4 * "x");
    "phi" := "phi" + "w0c_2_9_4" * SIN(4 * 0.4 * "x") + "w0d_2_9_4" * COS(4 * 0.4 * "x");
    "phi" := "phi" + "w0c_2_9_5" * SIN(5 * 0.4 * "x") + "w0d_2_9_5" * COS(5 * 0.4 * "x");
    "phi" := "phi" + "w0c_2_9_6" * SIN(6 * 0.4 * "x") + "w0d_2_9_6" * COS(6 * 0.4 * "x");
    "acc" := "acc" + "phi";
    "x" := "feat_10";
    "phi" := "w0b_2_10" * "x" / (1.0 + EXP(-"x"));
    "phi" := "phi" + "w0c_2_10_1" * SIN(1 * 0.4 * "x") + "w0d_2_10_1" * COS(1 * 0.4 * "x");
    "phi" := "phi" + "w0c_2_10_2" * SIN(2 * 0.4 * "x") + "w0d_2_10_2" * COS(2 * 0.4 * "x");
    "phi" := "phi" + "w0c_2_10_3" * SIN(3 * 0.4 * "x") + "w0d_2_10_3" * COS(3 * 0.4 * "x");
    "phi" := "phi" + "w0c_2_10_4" * SIN(4 * 0.4 * "x") + "w0d_2_10_4" * COS(4 * 0.4 * "x");
    "phi" := "phi" + "w0c_2_10_5" * SIN(5 * 0.4 * "x") + "w0d_2_10_5" * COS(5 * 0.4 * "x");
    "phi" := "phi" + "w0c_2_10_6" * SIN(6 * 0.4 * "x") + "w0d_2_10_6" * COS(6 * 0.4 * "x");
    "acc" := "acc" + "phi";
    "x" := "feat_11";
    "phi" := "w0b_2_11" * "x" / (1.0 + EXP(-"x"));
    "phi" := "phi" + "w0c_2_11_1" * SIN(1 * 0.4 * "x") + "w0d_2_11_1" * COS(1 * 0.4 * "x");
    "phi" := "phi" + "w0c_2_11_2" * SIN(2 * 0.4 * "x") + "w0d_2_11_2" * COS(2 * 0.4 * "x");
    "phi" := "phi" + "w0c_2_11_3" * SIN(3 * 0.4 * "x") + "w0d_2_11_3" * COS(3 * 0.4 * "x");
    "phi" := "phi" + "w0c_2_11_4" * SIN(4 * 0.4 * "x") + "w0d_2_11_4" * COS(4 * 0.4 * "x");
    "phi" := "phi" + "w0c_2_11_5" * SIN(5 * 0.4 * "x") + "w0d_2_11_5" * COS(5 * 0.4 * "x");
    "phi" := "phi" + "w0c_2_11_6" * SIN(6 * 0.4 * "x") + "w0d_2_11_6" * COS(6 * 0.4 * "x");
    "acc" := "acc" + "phi";
    "x" := "feat_12";
    "phi" := "w0b_2_12" * "x" / (1.0 + EXP(-"x"));
    "phi" := "phi" + "w0c_2_12_1" * SIN(1 * 0.4 * "x") + "w0d_2_12_1" * COS(1 * 0.4 * "x");
    "phi" := "phi" + "w0c_2_12_2" * SIN(2 * 0.4 * "x") + "w0d_2_12_2" * COS(2 * 0.4 * "x");
    "phi" := "phi" + "w0c_2_12_3" * SIN(3 * 0.4 * "x") + "w0d_2_12_3" * COS(3 * 0.4 * "x");
    "phi" := "phi" + "w0c_2_12_4" * SIN(4 * 0.4 * "x") + "w0d_2_12_4" * COS(4 * 0.4 * "x");
    "phi" := "phi" + "w0c_2_12_5" * SIN(5 * 0.4 * "x") + "w0d_2_12_5" * COS(5 * 0.4 * "x");
    "phi" := "phi" + "w0c_2_12_6" * SIN(6 * 0.4 * "x") + "w0d_2_12_6" * COS(6 * 0.4 * "x");
    "acc" := "acc" + "phi";
    "x" := "feat_13";
    "phi" := "w0b_2_13" * "x" / (1.0 + EXP(-"x"));
    "phi" := "phi" + "w0c_2_13_1" * SIN(1 * 0.4 * "x") + "w0d_2_13_1" * COS(1 * 0.4 * "x");
    "phi" := "phi" + "w0c_2_13_2" * SIN(2 * 0.4 * "x") + "w0d_2_13_2" * COS(2 * 0.4 * "x");
    "phi" := "phi" + "w0c_2_13_3" * SIN(3 * 0.4 * "x") + "w0d_2_13_3" * COS(3 * 0.4 * "x");
    "phi" := "phi" + "w0c_2_13_4" * SIN(4 * 0.4 * "x") + "w0d_2_13_4" * COS(4 * 0.4 * "x");
    "phi" := "phi" + "w0c_2_13_5" * SIN(5 * 0.4 * "x") + "w0d_2_13_5" * COS(5 * 0.4 * "x");
    "phi" := "phi" + "w0c_2_13_6" * SIN(6 * 0.4 * "x") + "w0d_2_13_6" * COS(6 * 0.4 * "x");
    "acc" := "acc" + "phi";
    "x" := "feat_14";
    "phi" := "w0b_2_14" * "x" / (1.0 + EXP(-"x"));
    "phi" := "phi" + "w0c_2_14_1" * SIN(1 * 0.4 * "x") + "w0d_2_14_1" * COS(1 * 0.4 * "x");
    "phi" := "phi" + "w0c_2_14_2" * SIN(2 * 0.4 * "x") + "w0d_2_14_2" * COS(2 * 0.4 * "x");
    "phi" := "phi" + "w0c_2_14_3" * SIN(3 * 0.4 * "x") + "w0d_2_14_3" * COS(3 * 0.4 * "x");
    "phi" := "phi" + "w0c_2_14_4" * SIN(4 * 0.4 * "x") + "w0d_2_14_4" * COS(4 * 0.4 * "x");
    "phi" := "phi" + "w0c_2_14_5" * SIN(5 * 0.4 * "x") + "w0d_2_14_5" * COS(5 * 0.4 * "x");
    "phi" := "phi" + "w0c_2_14_6" * SIN(6 * 0.4 * "x") + "w0d_2_14_6" * COS(6 * 0.4 * "x");
    "acc" := "acc" + "phi";
    "x" := "feat_15";
    "phi" := "w0b_2_15" * "x" / (1.0 + EXP(-"x"));
    "phi" := "phi" + "w0c_2_15_1" * SIN(1 * 0.4 * "x") + "w0d_2_15_1" * COS(1 * 0.4 * "x");
    "phi" := "phi" + "w0c_2_15_2" * SIN(2 * 0.4 * "x") + "w0d_2_15_2" * COS(2 * 0.4 * "x");
    "phi" := "phi" + "w0c_2_15_3" * SIN(3 * 0.4 * "x") + "w0d_2_15_3" * COS(3 * 0.4 * "x");
    "phi" := "phi" + "w0c_2_15_4" * SIN(4 * 0.4 * "x") + "w0d_2_15_4" * COS(4 * 0.4 * "x");
    "phi" := "phi" + "w0c_2_15_5" * SIN(5 * 0.4 * "x") + "w0d_2_15_5" * COS(5 * 0.4 * "x");
    "phi" := "phi" + "w0c_2_15_6" * SIN(6 * 0.4 * "x") + "w0d_2_15_6" * COS(6 * 0.4 * "x");
    "acc" := "acc" + "phi";
    "x" := "feat_16";
    "phi" := "w0b_2_16" * "x" / (1.0 + EXP(-"x"));
    "phi" := "phi" + "w0c_2_16_1" * SIN(1 * 0.4 * "x") + "w0d_2_16_1" * COS(1 * 0.4 * "x");
    "phi" := "phi" + "w0c_2_16_2" * SIN(2 * 0.4 * "x") + "w0d_2_16_2" * COS(2 * 0.4 * "x");
    "phi" := "phi" + "w0c_2_16_3" * SIN(3 * 0.4 * "x") + "w0d_2_16_3" * COS(3 * 0.4 * "x");
    "phi" := "phi" + "w0c_2_16_4" * SIN(4 * 0.4 * "x") + "w0d_2_16_4" * COS(4 * 0.4 * "x");
    "phi" := "phi" + "w0c_2_16_5" * SIN(5 * 0.4 * "x") + "w0d_2_16_5" * COS(5 * 0.4 * "x");
    "phi" := "phi" + "w0c_2_16_6" * SIN(6 * 0.4 * "x") + "w0d_2_16_6" * COS(6 * 0.4 * "x");
    "acc" := "acc" + "phi";
    "x" := "feat_17";
    "phi" := "w0b_2_17" * "x" / (1.0 + EXP(-"x"));
    "phi" := "phi" + "w0c_2_17_1" * SIN(1 * 0.4 * "x") + "w0d_2_17_1" * COS(1 * 0.4 * "x");
    "phi" := "phi" + "w0c_2_17_2" * SIN(2 * 0.4 * "x") + "w0d_2_17_2" * COS(2 * 0.4 * "x");
    "phi" := "phi" + "w0c_2_17_3" * SIN(3 * 0.4 * "x") + "w0d_2_17_3" * COS(3 * 0.4 * "x");
    "phi" := "phi" + "w0c_2_17_4" * SIN(4 * 0.4 * "x") + "w0d_2_17_4" * COS(4 * 0.4 * "x");
    "phi" := "phi" + "w0c_2_17_5" * SIN(5 * 0.4 * "x") + "w0d_2_17_5" * COS(5 * 0.4 * "x");
    "phi" := "phi" + "w0c_2_17_6" * SIN(6 * 0.4 * "x") + "w0d_2_17_6" * COS(6 * 0.4 * "x");
    "acc" := "acc" + "phi";
    "x" := "feat_18";
    "phi" := "w0b_2_18" * "x" / (1.0 + EXP(-"x"));
    "phi" := "phi" + "w0c_2_18_1" * SIN(1 * 0.4 * "x") + "w0d_2_18_1" * COS(1 * 0.4 * "x");
    "phi" := "phi" + "w0c_2_18_2" * SIN(2 * 0.4 * "x") + "w0d_2_18_2" * COS(2 * 0.4 * "x");
    "phi" := "phi" + "w0c_2_18_3" * SIN(3 * 0.4 * "x") + "w0d_2_18_3" * COS(3 * 0.4 * "x");
    "phi" := "phi" + "w0c_2_18_4" * SIN(4 * 0.4 * "x") + "w0d_2_18_4" * COS(4 * 0.4 * "x");
    "phi" := "phi" + "w0c_2_18_5" * SIN(5 * 0.4 * "x") + "w0d_2_18_5" * COS(5 * 0.4 * "x");
    "phi" := "phi" + "w0c_2_18_6" * SIN(6 * 0.4 * "x") + "w0d_2_18_6" * COS(6 * 0.4 * "x");
    "acc" := "acc" + "phi";
    "x" := "feat_19";
    "phi" := "w0b_2_19" * "x" / (1.0 + EXP(-"x"));
    "phi" := "phi" + "w0c_2_19_1" * SIN(1 * 0.4 * "x") + "w0d_2_19_1" * COS(1 * 0.4 * "x");
    "phi" := "phi" + "w0c_2_19_2" * SIN(2 * 0.4 * "x") + "w0d_2_19_2" * COS(2 * 0.4 * "x");
    "phi" := "phi" + "w0c_2_19_3" * SIN(3 * 0.4 * "x") + "w0d_2_19_3" * COS(3 * 0.4 * "x");
    "phi" := "phi" + "w0c_2_19_4" * SIN(4 * 0.4 * "x") + "w0d_2_19_4" * COS(4 * 0.4 * "x");
    "phi" := "phi" + "w0c_2_19_5" * SIN(5 * 0.4 * "x") + "w0d_2_19_5" * COS(5 * 0.4 * "x");
    "phi" := "phi" + "w0c_2_19_6" * SIN(6 * 0.4 * "x") + "w0d_2_19_6" * COS(6 * 0.4 * "x");
    "acc" := "acc" + "phi";
    "x" := "feat_20";
    "phi" := "w0b_2_20" * "x" / (1.0 + EXP(-"x"));
    "phi" := "phi" + "w0c_2_20_1" * SIN(1 * 0.4 * "x") + "w0d_2_20_1" * COS(1 * 0.4 * "x");
    "phi" := "phi" + "w0c_2_20_2" * SIN(2 * 0.4 * "x") + "w0d_2_20_2" * COS(2 * 0.4 * "x");
    "phi" := "phi" + "w0c_2_20_3" * SIN(3 * 0.4 * "x") + "w0d_2_20_3" * COS(3 * 0.4 * "x");
    "phi" := "phi" + "w0c_2_20_4" * SIN(4 * 0.4 * "x") + "w0d_2_20_4" * COS(4 * 0.4 * "x");
    "phi" := "phi" + "w0c_2_20_5" * SIN(5 * 0.4 * "x") + "w0d_2_20_5" * COS(5 * 0.4 * "x");
    "phi" := "phi" + "w0c_2_20_6" * SIN(6 * 0.4 * "x") + "w0d_2_20_6" * COS(6 * 0.4 * "x");
    "acc" := "acc" + "phi";
    "x" := "feat_21";
    "phi" := "w0b_2_21" * "x" / (1.0 + EXP(-"x"));
    "phi" := "phi" + "w0c_2_21_1" * SIN(1 * 0.4 * "x") + "w0d_2_21_1" * COS(1 * 0.4 * "x");
    "phi" := "phi" + "w0c_2_21_2" * SIN(2 * 0.4 * "x") + "w0d_2_21_2" * COS(2 * 0.4 * "x");
    "phi" := "phi" + "w0c_2_21_3" * SIN(3 * 0.4 * "x") + "w0d_2_21_3" * COS(3 * 0.4 * "x");
    "phi" := "phi" + "w0c_2_21_4" * SIN(4 * 0.4 * "x") + "w0d_2_21_4" * COS(4 * 0.4 * "x");
    "phi" := "phi" + "w0c_2_21_5" * SIN(5 * 0.4 * "x") + "w0d_2_21_5" * COS(5 * 0.4 * "x");
    "phi" := "phi" + "w0c_2_21_6" * SIN(6 * 0.4 * "x") + "w0d_2_21_6" * COS(6 * 0.4 * "x");
    "acc" := "acc" + "phi";
    "x" := "feat_22";
    "phi" := "w0b_2_22" * "x" / (1.0 + EXP(-"x"));
    "phi" := "phi" + "w0c_2_22_1" * SIN(1 * 0.4 * "x") + "w0d_2_22_1" * COS(1 * 0.4 * "x");
    "phi" := "phi" + "w0c_2_22_2" * SIN(2 * 0.4 * "x") + "w0d_2_22_2" * COS(2 * 0.4 * "x");
    "phi" := "phi" + "w0c_2_22_3" * SIN(3 * 0.4 * "x") + "w0d_2_22_3" * COS(3 * 0.4 * "x");
    "phi" := "phi" + "w0c_2_22_4" * SIN(4 * 0.4 * "x") + "w0d_2_22_4" * COS(4 * 0.4 * "x");
    "phi" := "phi" + "w0c_2_22_5" * SIN(5 * 0.4 * "x") + "w0d_2_22_5" * COS(5 * 0.4 * "x");
    "phi" := "phi" + "w0c_2_22_6" * SIN(6 * 0.4 * "x") + "w0d_2_22_6" * COS(6 * 0.4 * "x");
    "acc" := "acc" + "phi";
    "x" := "feat_23";
    "phi" := "w0b_2_23" * "x" / (1.0 + EXP(-"x"));
    "phi" := "phi" + "w0c_2_23_1" * SIN(1 * 0.4 * "x") + "w0d_2_23_1" * COS(1 * 0.4 * "x");
    "phi" := "phi" + "w0c_2_23_2" * SIN(2 * 0.4 * "x") + "w0d_2_23_2" * COS(2 * 0.4 * "x");
    "phi" := "phi" + "w0c_2_23_3" * SIN(3 * 0.4 * "x") + "w0d_2_23_3" * COS(3 * 0.4 * "x");
    "phi" := "phi" + "w0c_2_23_4" * SIN(4 * 0.4 * "x") + "w0d_2_23_4" * COS(4 * 0.4 * "x");
    "phi" := "phi" + "w0c_2_23_5" * SIN(5 * 0.4 * "x") + "w0d_2_23_5" * COS(5 * 0.4 * "x");
    "phi" := "phi" + "w0c_2_23_6" * SIN(6 * 0.4 * "x") + "w0d_2_23_6" * COS(6 * 0.4 * "x");
    "acc" := "acc" + "phi";
    "x" := "feat_24";
    "phi" := "w0b_2_24" * "x" / (1.0 + EXP(-"x"));
    "phi" := "phi" + "w0c_2_24_1" * SIN(1 * 0.4 * "x") + "w0d_2_24_1" * COS(1 * 0.4 * "x");
    "phi" := "phi" + "w0c_2_24_2" * SIN(2 * 0.4 * "x") + "w0d_2_24_2" * COS(2 * 0.4 * "x");
    "phi" := "phi" + "w0c_2_24_3" * SIN(3 * 0.4 * "x") + "w0d_2_24_3" * COS(3 * 0.4 * "x");
    "phi" := "phi" + "w0c_2_24_4" * SIN(4 * 0.4 * "x") + "w0d_2_24_4" * COS(4 * 0.4 * "x");
    "phi" := "phi" + "w0c_2_24_5" * SIN(5 * 0.4 * "x") + "w0d_2_24_5" * COS(5 * 0.4 * "x");
    "phi" := "phi" + "w0c_2_24_6" * SIN(6 * 0.4 * "x") + "w0d_2_24_6" * COS(6 * 0.4 * "x");
    "acc" := "acc" + "phi";
    "x" := "feat_25";
    "phi" := "w0b_2_25" * "x" / (1.0 + EXP(-"x"));
    "phi" := "phi" + "w0c_2_25_1" * SIN(1 * 0.4 * "x") + "w0d_2_25_1" * COS(1 * 0.4 * "x");
    "phi" := "phi" + "w0c_2_25_2" * SIN(2 * 0.4 * "x") + "w0d_2_25_2" * COS(2 * 0.4 * "x");
    "phi" := "phi" + "w0c_2_25_3" * SIN(3 * 0.4 * "x") + "w0d_2_25_3" * COS(3 * 0.4 * "x");
    "phi" := "phi" + "w0c_2_25_4" * SIN(4 * 0.4 * "x") + "w0d_2_25_4" * COS(4 * 0.4 * "x");
    "phi" := "phi" + "w0c_2_25_5" * SIN(5 * 0.4 * "x") + "w0d_2_25_5" * COS(5 * 0.4 * "x");
    "phi" := "phi" + "w0c_2_25_6" * SIN(6 * 0.4 * "x") + "w0d_2_25_6" * COS(6 * 0.4 * "x");
    "acc" := "acc" + "phi";
    "x" := "feat_26";
    "phi" := "w0b_2_26" * "x" / (1.0 + EXP(-"x"));
    "phi" := "phi" + "w0c_2_26_1" * SIN(1 * 0.4 * "x") + "w0d_2_26_1" * COS(1 * 0.4 * "x");
    "phi" := "phi" + "w0c_2_26_2" * SIN(2 * 0.4 * "x") + "w0d_2_26_2" * COS(2 * 0.4 * "x");
    "phi" := "phi" + "w0c_2_26_3" * SIN(3 * 0.4 * "x") + "w0d_2_26_3" * COS(3 * 0.4 * "x");
    "phi" := "phi" + "w0c_2_26_4" * SIN(4 * 0.4 * "x") + "w0d_2_26_4" * COS(4 * 0.4 * "x");
    "phi" := "phi" + "w0c_2_26_5" * SIN(5 * 0.4 * "x") + "w0d_2_26_5" * COS(5 * 0.4 * "x");
    "phi" := "phi" + "w0c_2_26_6" * SIN(6 * 0.4 * "x") + "w0d_2_26_6" * COS(6 * 0.4 * "x");
    "acc" := "acc" + "phi";
    "x" := "feat_27";
    "phi" := "w0b_2_27" * "x" / (1.0 + EXP(-"x"));
    "phi" := "phi" + "w0c_2_27_1" * SIN(1 * 0.4 * "x") + "w0d_2_27_1" * COS(1 * 0.4 * "x");
    "phi" := "phi" + "w0c_2_27_2" * SIN(2 * 0.4 * "x") + "w0d_2_27_2" * COS(2 * 0.4 * "x");
    "phi" := "phi" + "w0c_2_27_3" * SIN(3 * 0.4 * "x") + "w0d_2_27_3" * COS(3 * 0.4 * "x");
    "phi" := "phi" + "w0c_2_27_4" * SIN(4 * 0.4 * "x") + "w0d_2_27_4" * COS(4 * 0.4 * "x");
    "phi" := "phi" + "w0c_2_27_5" * SIN(5 * 0.4 * "x") + "w0d_2_27_5" * COS(5 * 0.4 * "x");
    "phi" := "phi" + "w0c_2_27_6" * SIN(6 * 0.4 * "x") + "w0d_2_27_6" * COS(6 * 0.4 * "x");
    "acc" := "acc" + "phi";
    "x" := "feat_28";
    "phi" := "w0b_2_28" * "x" / (1.0 + EXP(-"x"));
    "phi" := "phi" + "w0c_2_28_1" * SIN(1 * 0.4 * "x") + "w0d_2_28_1" * COS(1 * 0.4 * "x");
    "phi" := "phi" + "w0c_2_28_2" * SIN(2 * 0.4 * "x") + "w0d_2_28_2" * COS(2 * 0.4 * "x");
    "phi" := "phi" + "w0c_2_28_3" * SIN(3 * 0.4 * "x") + "w0d_2_28_3" * COS(3 * 0.4 * "x");
    "phi" := "phi" + "w0c_2_28_4" * SIN(4 * 0.4 * "x") + "w0d_2_28_4" * COS(4 * 0.4 * "x");
    "phi" := "phi" + "w0c_2_28_5" * SIN(5 * 0.4 * "x") + "w0d_2_28_5" * COS(5 * 0.4 * "x");
    "phi" := "phi" + "w0c_2_28_6" * SIN(6 * 0.4 * "x") + "w0d_2_28_6" * COS(6 * 0.4 * "x");
    "acc" := "acc" + "phi";
    "h1_2" := "acc" + "b0_2";
    "acc" := 0.0;
    "x" := "feat_1";
    "phi" := "w0b_3_1" * "x" / (1.0 + EXP(-"x"));
    "phi" := "phi" + "w0c_3_1_1" * SIN(1 * 0.4 * "x") + "w0d_3_1_1" * COS(1 * 0.4 * "x");
    "phi" := "phi" + "w0c_3_1_2" * SIN(2 * 0.4 * "x") + "w0d_3_1_2" * COS(2 * 0.4 * "x");
    "phi" := "phi" + "w0c_3_1_3" * SIN(3 * 0.4 * "x") + "w0d_3_1_3" * COS(3 * 0.4 * "x");
    "phi" := "phi" + "w0c_3_1_4" * SIN(4 * 0.4 * "x") + "w0d_3_1_4" * COS(4 * 0.4 * "x");
    "phi" := "phi" + "w0c_3_1_5" * SIN(5 * 0.4 * "x") + "w0d_3_1_5" * COS(5 * 0.4 * "x");
    "phi" := "phi" + "w0c_3_1_6" * SIN(6 * 0.4 * "x") + "w0d_3_1_6" * COS(6 * 0.4 * "x");
    "acc" := "acc" + "phi";
    "x" := "feat_2";
    "phi" := "w0b_3_2" * "x" / (1.0 + EXP(-"x"));
    "phi" := "phi" + "w0c_3_2_1" * SIN(1 * 0.4 * "x") + "w0d_3_2_1" * COS(1 * 0.4 * "x");
    "phi" := "phi" + "w0c_3_2_2" * SIN(2 * 0.4 * "x") + "w0d_3_2_2" * COS(2 * 0.4 * "x");
    "phi" := "phi" + "w0c_3_2_3" * SIN(3 * 0.4 * "x") + "w0d_3_2_3" * COS(3 * 0.4 * "x");
    "phi" := "phi" + "w0c_3_2_4" * SIN(4 * 0.4 * "x") + "w0d_3_2_4" * COS(4 * 0.4 * "x");
    "phi" := "phi" + "w0c_3_2_5" * SIN(5 * 0.4 * "x") + "w0d_3_2_5" * COS(5 * 0.4 * "x");
    "phi" := "phi" + "w0c_3_2_6" * SIN(6 * 0.4 * "x") + "w0d_3_2_6" * COS(6 * 0.4 * "x");
    "acc" := "acc" + "phi";
    "x" := "feat_3";
    "phi" := "w0b_3_3" * "x" / (1.0 + EXP(-"x"));
    "phi" := "phi" + "w0c_3_3_1" * SIN(1 * 0.4 * "x") + "w0d_3_3_1" * COS(1 * 0.4 * "x");
    "phi" := "phi" + "w0c_3_3_2" * SIN(2 * 0.4 * "x") + "w0d_3_3_2" * COS(2 * 0.4 * "x");
    "phi" := "phi" + "w0c_3_3_3" * SIN(3 * 0.4 * "x") + "w0d_3_3_3" * COS(3 * 0.4 * "x");
    "phi" := "phi" + "w0c_3_3_4" * SIN(4 * 0.4 * "x") + "w0d_3_3_4" * COS(4 * 0.4 * "x");
    "phi" := "phi" + "w0c_3_3_5" * SIN(5 * 0.4 * "x") + "w0d_3_3_5" * COS(5 * 0.4 * "x");
    "phi" := "phi" + "w0c_3_3_6" * SIN(6 * 0.4 * "x") + "w0d_3_3_6" * COS(6 * 0.4 * "x");
    "acc" := "acc" + "phi";
    "x" := "feat_4";
    "phi" := "w0b_3_4" * "x" / (1.0 + EXP(-"x"));
    "phi" := "phi" + "w0c_3_4_1" * SIN(1 * 0.4 * "x") + "w0d_3_4_1" * COS(1 * 0.4 * "x");
    "phi" := "phi" + "w0c_3_4_2" * SIN(2 * 0.4 * "x") + "w0d_3_4_2" * COS(2 * 0.4 * "x");
    "phi" := "phi" + "w0c_3_4_3" * SIN(3 * 0.4 * "x") + "w0d_3_4_3" * COS(3 * 0.4 * "x");
    "phi" := "phi" + "w0c_3_4_4" * SIN(4 * 0.4 * "x") + "w0d_3_4_4" * COS(4 * 0.4 * "x");
    "phi" := "phi" + "w0c_3_4_5" * SIN(5 * 0.4 * "x") + "w0d_3_4_5" * COS(5 * 0.4 * "x");
    "phi" := "phi" + "w0c_3_4_6" * SIN(6 * 0.4 * "x") + "w0d_3_4_6" * COS(6 * 0.4 * "x");
    "acc" := "acc" + "phi";
    "x" := "feat_5";
    "phi" := "w0b_3_5" * "x" / (1.0 + EXP(-"x"));
    "phi" := "phi" + "w0c_3_5_1" * SIN(1 * 0.4 * "x") + "w0d_3_5_1" * COS(1 * 0.4 * "x");
    "phi" := "phi" + "w0c_3_5_2" * SIN(2 * 0.4 * "x") + "w0d_3_5_2" * COS(2 * 0.4 * "x");
    "phi" := "phi" + "w0c_3_5_3" * SIN(3 * 0.4 * "x") + "w0d_3_5_3" * COS(3 * 0.4 * "x");
    "phi" := "phi" + "w0c_3_5_4" * SIN(4 * 0.4 * "x") + "w0d_3_5_4" * COS(4 * 0.4 * "x");
    "phi" := "phi" + "w0c_3_5_5" * SIN(5 * 0.4 * "x") + "w0d_3_5_5" * COS(5 * 0.4 * "x");
    "phi" := "phi" + "w0c_3_5_6" * SIN(6 * 0.4 * "x") + "w0d_3_5_6" * COS(6 * 0.4 * "x");
    "acc" := "acc" + "phi";
    "x" := "feat_6";
    "phi" := "w0b_3_6" * "x" / (1.0 + EXP(-"x"));
    "phi" := "phi" + "w0c_3_6_1" * SIN(1 * 0.4 * "x") + "w0d_3_6_1" * COS(1 * 0.4 * "x");
    "phi" := "phi" + "w0c_3_6_2" * SIN(2 * 0.4 * "x") + "w0d_3_6_2" * COS(2 * 0.4 * "x");
    "phi" := "phi" + "w0c_3_6_3" * SIN(3 * 0.4 * "x") + "w0d_3_6_3" * COS(3 * 0.4 * "x");
    "phi" := "phi" + "w0c_3_6_4" * SIN(4 * 0.4 * "x") + "w0d_3_6_4" * COS(4 * 0.4 * "x");
    "phi" := "phi" + "w0c_3_6_5" * SIN(5 * 0.4 * "x") + "w0d_3_6_5" * COS(5 * 0.4 * "x");
    "phi" := "phi" + "w0c_3_6_6" * SIN(6 * 0.4 * "x") + "w0d_3_6_6" * COS(6 * 0.4 * "x");
    "acc" := "acc" + "phi";
    "x" := "feat_7";
    "phi" := "w0b_3_7" * "x" / (1.0 + EXP(-"x"));
    "phi" := "phi" + "w0c_3_7_1" * SIN(1 * 0.4 * "x") + "w0d_3_7_1" * COS(1 * 0.4 * "x");
    "phi" := "phi" + "w0c_3_7_2" * SIN(2 * 0.4 * "x") + "w0d_3_7_2" * COS(2 * 0.4 * "x");
    "phi" := "phi" + "w0c_3_7_3" * SIN(3 * 0.4 * "x") + "w0d_3_7_3" * COS(3 * 0.4 * "x");
    "phi" := "phi" + "w0c_3_7_4" * SIN(4 * 0.4 * "x") + "w0d_3_7_4" * COS(4 * 0.4 * "x");
    "phi" := "phi" + "w0c_3_7_5" * SIN(5 * 0.4 * "x") + "w0d_3_7_5" * COS(5 * 0.4 * "x");
    "phi" := "phi" + "w0c_3_7_6" * SIN(6 * 0.4 * "x") + "w0d_3_7_6" * COS(6 * 0.4 * "x");
    "acc" := "acc" + "phi";
    "x" := "feat_8";
    "phi" := "w0b_3_8" * "x" / (1.0 + EXP(-"x"));
    "phi" := "phi" + "w0c_3_8_1" * SIN(1 * 0.4 * "x") + "w0d_3_8_1" * COS(1 * 0.4 * "x");
    "phi" := "phi" + "w0c_3_8_2" * SIN(2 * 0.4 * "x") + "w0d_3_8_2" * COS(2 * 0.4 * "x");
    "phi" := "phi" + "w0c_3_8_3" * SIN(3 * 0.4 * "x") + "w0d_3_8_3" * COS(3 * 0.4 * "x");
    "phi" := "phi" + "w0c_3_8_4" * SIN(4 * 0.4 * "x") + "w0d_3_8_4" * COS(4 * 0.4 * "x");
    "phi" := "phi" + "w0c_3_8_5" * SIN(5 * 0.4 * "x") + "w0d_3_8_5" * COS(5 * 0.4 * "x");
    "phi" := "phi" + "w0c_3_8_6" * SIN(6 * 0.4 * "x") + "w0d_3_8_6" * COS(6 * 0.4 * "x");
    "acc" := "acc" + "phi";
    "x" := "feat_9";
    "phi" := "w0b_3_9" * "x" / (1.0 + EXP(-"x"));
    "phi" := "phi" + "w0c_3_9_1" * SIN(1 * 0.4 * "x") + "w0d_3_9_1" * COS(1 * 0.4 * "x");
    "phi" := "phi" + "w0c_3_9_2" * SIN(2 * 0.4 * "x") + "w0d_3_9_2" * COS(2 * 0.4 * "x");
    "phi" := "phi" + "w0c_3_9_3" * SIN(3 * 0.4 * "x") + "w0d_3_9_3" * COS(3 * 0.4 * "x");
    "phi" := "phi" + "w0c_3_9_4" * SIN(4 * 0.4 * "x") + "w0d_3_9_4" * COS(4 * 0.4 * "x");
    "phi" := "phi" + "w0c_3_9_5" * SIN(5 * 0.4 * "x") + "w0d_3_9_5" * COS(5 * 0.4 * "x");
    "phi" := "phi" + "w0c_3_9_6" * SIN(6 * 0.4 * "x") + "w0d_3_9_6" * COS(6 * 0.4 * "x");
    "acc" := "acc" + "phi";
    "x" := "feat_10";
    "phi" := "w0b_3_10" * "x" / (1.0 + EXP(-"x"));
    "phi" := "phi" + "w0c_3_10_1" * SIN(1 * 0.4 * "x") + "w0d_3_10_1" * COS(1 * 0.4 * "x");
    "phi" := "phi" + "w0c_3_10_2" * SIN(2 * 0.4 * "x") + "w0d_3_10_2" * COS(2 * 0.4 * "x");
    "phi" := "phi" + "w0c_3_10_3" * SIN(3 * 0.4 * "x") + "w0d_3_10_3" * COS(3 * 0.4 * "x");
    "phi" := "phi" + "w0c_3_10_4" * SIN(4 * 0.4 * "x") + "w0d_3_10_4" * COS(4 * 0.4 * "x");
    "phi" := "phi" + "w0c_3_10_5" * SIN(5 * 0.4 * "x") + "w0d_3_10_5" * COS(5 * 0.4 * "x");
    "phi" := "phi" + "w0c_3_10_6" * SIN(6 * 0.4 * "x") + "w0d_3_10_6" * COS(6 * 0.4 * "x");
    "acc" := "acc" + "phi";
    "x" := "feat_11";
    "phi" := "w0b_3_11" * "x" / (1.0 + EXP(-"x"));
    "phi" := "phi" + "w0c_3_11_1" * SIN(1 * 0.4 * "x") + "w0d_3_11_1" * COS(1 * 0.4 * "x");
    "phi" := "phi" + "w0c_3_11_2" * SIN(2 * 0.4 * "x") + "w0d_3_11_2" * COS(2 * 0.4 * "x");
    "phi" := "phi" + "w0c_3_11_3" * SIN(3 * 0.4 * "x") + "w0d_3_11_3" * COS(3 * 0.4 * "x");
    "phi" := "phi" + "w0c_3_11_4" * SIN(4 * 0.4 * "x") + "w0d_3_11_4" * COS(4 * 0.4 * "x");
    "phi" := "phi" + "w0c_3_11_5" * SIN(5 * 0.4 * "x") + "w0d_3_11_5" * COS(5 * 0.4 * "x");
    "phi" := "phi" + "w0c_3_11_6" * SIN(6 * 0.4 * "x") + "w0d_3_11_6" * COS(6 * 0.4 * "x");
    "acc" := "acc" + "phi";
    "x" := "feat_12";
    "phi" := "w0b_3_12" * "x" / (1.0 + EXP(-"x"));
    "phi" := "phi" + "w0c_3_12_1" * SIN(1 * 0.4 * "x") + "w0d_3_12_1" * COS(1 * 0.4 * "x");
    "phi" := "phi" + "w0c_3_12_2" * SIN(2 * 0.4 * "x") + "w0d_3_12_2" * COS(2 * 0.4 * "x");
    "phi" := "phi" + "w0c_3_12_3" * SIN(3 * 0.4 * "x") + "w0d_3_12_3" * COS(3 * 0.4 * "x");
    "phi" := "phi" + "w0c_3_12_4" * SIN(4 * 0.4 * "x") + "w0d_3_12_4" * COS(4 * 0.4 * "x");
    "phi" := "phi" + "w0c_3_12_5" * SIN(5 * 0.4 * "x") + "w0d_3_12_5" * COS(5 * 0.4 * "x");
    "phi" := "phi" + "w0c_3_12_6" * SIN(6 * 0.4 * "x") + "w0d_3_12_6" * COS(6 * 0.4 * "x");
    "acc" := "acc" + "phi";
    "x" := "feat_13";
    "phi" := "w0b_3_13" * "x" / (1.0 + EXP(-"x"));
    "phi" := "phi" + "w0c_3_13_1" * SIN(1 * 0.4 * "x") + "w0d_3_13_1" * COS(1 * 0.4 * "x");
    "phi" := "phi" + "w0c_3_13_2" * SIN(2 * 0.4 * "x") + "w0d_3_13_2" * COS(2 * 0.4 * "x");
    "phi" := "phi" + "w0c_3_13_3" * SIN(3 * 0.4 * "x") + "w0d_3_13_3" * COS(3 * 0.4 * "x");
    "phi" := "phi" + "w0c_3_13_4" * SIN(4 * 0.4 * "x") + "w0d_3_13_4" * COS(4 * 0.4 * "x");
    "phi" := "phi" + "w0c_3_13_5" * SIN(5 * 0.4 * "x") + "w0d_3_13_5" * COS(5 * 0.4 * "x");
    "phi" := "phi" + "w0c_3_13_6" * SIN(6 * 0.4 * "x") + "w0d_3_13_6" * COS(6 * 0.4 * "x");
    "acc" := "acc" + "phi";
    "x" := "feat_14";
    "phi" := "w0b_3_14" * "x" / (1.0 + EXP(-"x"));
    "phi" := "phi" + "w0c_3_14_1" * SIN(1 * 0.4 * "x") + "w0d_3_14_1" * COS(1 * 0.4 * "x");
    "phi" := "phi" + "w0c_3_14_2" * SIN(2 * 0.4 * "x") + "w0d_3_14_2" * COS(2 * 0.4 * "x");
    "phi" := "phi" + "w0c_3_14_3" * SIN(3 * 0.4 * "x") + "w0d_3_14_3" * COS(3 * 0.4 * "x");
    "phi" := "phi" + "w0c_3_14_4" * SIN(4 * 0.4 * "x") + "w0d_3_14_4" * COS(4 * 0.4 * "x");
    "phi" := "phi" + "w0c_3_14_5" * SIN(5 * 0.4 * "x") + "w0d_3_14_5" * COS(5 * 0.4 * "x");
    "phi" := "phi" + "w0c_3_14_6" * SIN(6 * 0.4 * "x") + "w0d_3_14_6" * COS(6 * 0.4 * "x");
    "acc" := "acc" + "phi";
    "x" := "feat_15";
    "phi" := "w0b_3_15" * "x" / (1.0 + EXP(-"x"));
    "phi" := "phi" + "w0c_3_15_1" * SIN(1 * 0.4 * "x") + "w0d_3_15_1" * COS(1 * 0.4 * "x");
    "phi" := "phi" + "w0c_3_15_2" * SIN(2 * 0.4 * "x") + "w0d_3_15_2" * COS(2 * 0.4 * "x");
    "phi" := "phi" + "w0c_3_15_3" * SIN(3 * 0.4 * "x") + "w0d_3_15_3" * COS(3 * 0.4 * "x");
    "phi" := "phi" + "w0c_3_15_4" * SIN(4 * 0.4 * "x") + "w0d_3_15_4" * COS(4 * 0.4 * "x");
    "phi" := "phi" + "w0c_3_15_5" * SIN(5 * 0.4 * "x") + "w0d_3_15_5" * COS(5 * 0.4 * "x");
    "phi" := "phi" + "w0c_3_15_6" * SIN(6 * 0.4 * "x") + "w0d_3_15_6" * COS(6 * 0.4 * "x");
    "acc" := "acc" + "phi";
    "x" := "feat_16";
    "phi" := "w0b_3_16" * "x" / (1.0 + EXP(-"x"));
    "phi" := "phi" + "w0c_3_16_1" * SIN(1 * 0.4 * "x") + "w0d_3_16_1" * COS(1 * 0.4 * "x");
    "phi" := "phi" + "w0c_3_16_2" * SIN(2 * 0.4 * "x") + "w0d_3_16_2" * COS(2 * 0.4 * "x");
    "phi" := "phi" + "w0c_3_16_3" * SIN(3 * 0.4 * "x") + "w0d_3_16_3" * COS(3 * 0.4 * "x");
    "phi" := "phi" + "w0c_3_16_4" * SIN(4 * 0.4 * "x") + "w0d_3_16_4" * COS(4 * 0.4 * "x");
    "phi" := "phi" + "w0c_3_16_5" * SIN(5 * 0.4 * "x") + "w0d_3_16_5" * COS(5 * 0.4 * "x");
    "phi" := "phi" + "w0c_3_16_6" * SIN(6 * 0.4 * "x") + "w0d_3_16_6" * COS(6 * 0.4 * "x");
    "acc" := "acc" + "phi";
    "x" := "feat_17";
    "phi" := "w0b_3_17" * "x" / (1.0 + EXP(-"x"));
    "phi" := "phi" + "w0c_3_17_1" * SIN(1 * 0.4 * "x") + "w0d_3_17_1" * COS(1 * 0.4 * "x");
    "phi" := "phi" + "w0c_3_17_2" * SIN(2 * 0.4 * "x") + "w0d_3_17_2" * COS(2 * 0.4 * "x");
    "phi" := "phi" + "w0c_3_17_3" * SIN(3 * 0.4 * "x") + "w0d_3_17_3" * COS(3 * 0.4 * "x");
    "phi" := "phi" + "w0c_3_17_4" * SIN(4 * 0.4 * "x") + "w0d_3_17_4" * COS(4 * 0.4 * "x");
    "phi" := "phi" + "w0c_3_17_5" * SIN(5 * 0.4 * "x") + "w0d_3_17_5" * COS(5 * 0.4 * "x");
    "phi" := "phi" + "w0c_3_17_6" * SIN(6 * 0.4 * "x") + "w0d_3_17_6" * COS(6 * 0.4 * "x");
    "acc" := "acc" + "phi";
    "x" := "feat_18";
    "phi" := "w0b_3_18" * "x" / (1.0 + EXP(-"x"));
    "phi" := "phi" + "w0c_3_18_1" * SIN(1 * 0.4 * "x") + "w0d_3_18_1" * COS(1 * 0.4 * "x");
    "phi" := "phi" + "w0c_3_18_2" * SIN(2 * 0.4 * "x") + "w0d_3_18_2" * COS(2 * 0.4 * "x");
    "phi" := "phi" + "w0c_3_18_3" * SIN(3 * 0.4 * "x") + "w0d_3_18_3" * COS(3 * 0.4 * "x");
    "phi" := "phi" + "w0c_3_18_4" * SIN(4 * 0.4 * "x") + "w0d_3_18_4" * COS(4 * 0.4 * "x");
    "phi" := "phi" + "w0c_3_18_5" * SIN(5 * 0.4 * "x") + "w0d_3_18_5" * COS(5 * 0.4 * "x");
    "phi" := "phi" + "w0c_3_18_6" * SIN(6 * 0.4 * "x") + "w0d_3_18_6" * COS(6 * 0.4 * "x");
    "acc" := "acc" + "phi";
    "x" := "feat_19";
    "phi" := "w0b_3_19" * "x" / (1.0 + EXP(-"x"));
    "phi" := "phi" + "w0c_3_19_1" * SIN(1 * 0.4 * "x") + "w0d_3_19_1" * COS(1 * 0.4 * "x");
    "phi" := "phi" + "w0c_3_19_2" * SIN(2 * 0.4 * "x") + "w0d_3_19_2" * COS(2 * 0.4 * "x");
    "phi" := "phi" + "w0c_3_19_3" * SIN(3 * 0.4 * "x") + "w0d_3_19_3" * COS(3 * 0.4 * "x");
    "phi" := "phi" + "w0c_3_19_4" * SIN(4 * 0.4 * "x") + "w0d_3_19_4" * COS(4 * 0.4 * "x");
    "phi" := "phi" + "w0c_3_19_5" * SIN(5 * 0.4 * "x") + "w0d_3_19_5" * COS(5 * 0.4 * "x");
    "phi" := "phi" + "w0c_3_19_6" * SIN(6 * 0.4 * "x") + "w0d_3_19_6" * COS(6 * 0.4 * "x");
    "acc" := "acc" + "phi";
    "x" := "feat_20";
    "phi" := "w0b_3_20" * "x" / (1.0 + EXP(-"x"));
    "phi" := "phi" + "w0c_3_20_1" * SIN(1 * 0.4 * "x") + "w0d_3_20_1" * COS(1 * 0.4 * "x");
    "phi" := "phi" + "w0c_3_20_2" * SIN(2 * 0.4 * "x") + "w0d_3_20_2" * COS(2 * 0.4 * "x");
    "phi" := "phi" + "w0c_3_20_3" * SIN(3 * 0.4 * "x") + "w0d_3_20_3" * COS(3 * 0.4 * "x");
    "phi" := "phi" + "w0c_3_20_4" * SIN(4 * 0.4 * "x") + "w0d_3_20_4" * COS(4 * 0.4 * "x");
    "phi" := "phi" + "w0c_3_20_5" * SIN(5 * 0.4 * "x") + "w0d_3_20_5" * COS(5 * 0.4 * "x");
    "phi" := "phi" + "w0c_3_20_6" * SIN(6 * 0.4 * "x") + "w0d_3_20_6" * COS(6 * 0.4 * "x");
    "acc" := "acc" + "phi";
    "x" := "feat_21";
    "phi" := "w0b_3_21" * "x" / (1.0 + EXP(-"x"));
    "phi" := "phi" + "w0c_3_21_1" * SIN(1 * 0.4 * "x") + "w0d_3_21_1" * COS(1 * 0.4 * "x");
    "phi" := "phi" + "w0c_3_21_2" * SIN(2 * 0.4 * "x") + "w0d_3_21_2" * COS(2 * 0.4 * "x");
    "phi" := "phi" + "w0c_3_21_3" * SIN(3 * 0.4 * "x") + "w0d_3_21_3" * COS(3 * 0.4 * "x");
    "phi" := "phi" + "w0c_3_21_4" * SIN(4 * 0.4 * "x") + "w0d_3_21_4" * COS(4 * 0.4 * "x");
    "phi" := "phi" + "w0c_3_21_5" * SIN(5 * 0.4 * "x") + "w0d_3_21_5" * COS(5 * 0.4 * "x");
    "phi" := "phi" + "w0c_3_21_6" * SIN(6 * 0.4 * "x") + "w0d_3_21_6" * COS(6 * 0.4 * "x");
    "acc" := "acc" + "phi";
    "x" := "feat_22";
    "phi" := "w0b_3_22" * "x" / (1.0 + EXP(-"x"));
    "phi" := "phi" + "w0c_3_22_1" * SIN(1 * 0.4 * "x") + "w0d_3_22_1" * COS(1 * 0.4 * "x");
    "phi" := "phi" + "w0c_3_22_2" * SIN(2 * 0.4 * "x") + "w0d_3_22_2" * COS(2 * 0.4 * "x");
    "phi" := "phi" + "w0c_3_22_3" * SIN(3 * 0.4 * "x") + "w0d_3_22_3" * COS(3 * 0.4 * "x");
    "phi" := "phi" + "w0c_3_22_4" * SIN(4 * 0.4 * "x") + "w0d_3_22_4" * COS(4 * 0.4 * "x");
    "phi" := "phi" + "w0c_3_22_5" * SIN(5 * 0.4 * "x") + "w0d_3_22_5" * COS(5 * 0.4 * "x");
    "phi" := "phi" + "w0c_3_22_6" * SIN(6 * 0.4 * "x") + "w0d_3_22_6" * COS(6 * 0.4 * "x");
    "acc" := "acc" + "phi";
    "x" := "feat_23";
    "phi" := "w0b_3_23" * "x" / (1.0 + EXP(-"x"));
    "phi" := "phi" + "w0c_3_23_1" * SIN(1 * 0.4 * "x") + "w0d_3_23_1" * COS(1 * 0.4 * "x");
    "phi" := "phi" + "w0c_3_23_2" * SIN(2 * 0.4 * "x") + "w0d_3_23_2" * COS(2 * 0.4 * "x");
    "phi" := "phi" + "w0c_3_23_3" * SIN(3 * 0.4 * "x") + "w0d_3_23_3" * COS(3 * 0.4 * "x");
    "phi" := "phi" + "w0c_3_23_4" * SIN(4 * 0.4 * "x") + "w0d_3_23_4" * COS(4 * 0.4 * "x");
    "phi" := "phi" + "w0c_3_23_5" * SIN(5 * 0.4 * "x") + "w0d_3_23_5" * COS(5 * 0.4 * "x");
    "phi" := "phi" + "w0c_3_23_6" * SIN(6 * 0.4 * "x") + "w0d_3_23_6" * COS(6 * 0.4 * "x");
    "acc" := "acc" + "phi";
    "x" := "feat_24";
    "phi" := "w0b_3_24" * "x" / (1.0 + EXP(-"x"));
    "phi" := "phi" + "w0c_3_24_1" * SIN(1 * 0.4 * "x") + "w0d_3_24_1" * COS(1 * 0.4 * "x");
    "phi" := "phi" + "w0c_3_24_2" * SIN(2 * 0.4 * "x") + "w0d_3_24_2" * COS(2 * 0.4 * "x");
    "phi" := "phi" + "w0c_3_24_3" * SIN(3 * 0.4 * "x") + "w0d_3_24_3" * COS(3 * 0.4 * "x");
    "phi" := "phi" + "w0c_3_24_4" * SIN(4 * 0.4 * "x") + "w0d_3_24_4" * COS(4 * 0.4 * "x");
    "phi" := "phi" + "w0c_3_24_5" * SIN(5 * 0.4 * "x") + "w0d_3_24_5" * COS(5 * 0.4 * "x");
    "phi" := "phi" + "w0c_3_24_6" * SIN(6 * 0.4 * "x") + "w0d_3_24_6" * COS(6 * 0.4 * "x");
    "acc" := "acc" + "phi";
    "x" := "feat_25";
    "phi" := "w0b_3_25" * "x" / (1.0 + EXP(-"x"));
    "phi" := "phi" + "w0c_3_25_1" * SIN(1 * 0.4 * "x") + "w0d_3_25_1" * COS(1 * 0.4 * "x");
    "phi" := "phi" + "w0c_3_25_2" * SIN(2 * 0.4 * "x") + "w0d_3_25_2" * COS(2 * 0.4 * "x");
    "phi" := "phi" + "w0c_3_25_3" * SIN(3 * 0.4 * "x") + "w0d_3_25_3" * COS(3 * 0.4 * "x");
    "phi" := "phi" + "w0c_3_25_4" * SIN(4 * 0.4 * "x") + "w0d_3_25_4" * COS(4 * 0.4 * "x");
    "phi" := "phi" + "w0c_3_25_5" * SIN(5 * 0.4 * "x") + "w0d_3_25_5" * COS(5 * 0.4 * "x");
    "phi" := "phi" + "w0c_3_25_6" * SIN(6 * 0.4 * "x") + "w0d_3_25_6" * COS(6 * 0.4 * "x");
    "acc" := "acc" + "phi";
    "x" := "feat_26";
    "phi" := "w0b_3_26" * "x" / (1.0 + EXP(-"x"));
    "phi" := "phi" + "w0c_3_26_1" * SIN(1 * 0.4 * "x") + "w0d_3_26_1" * COS(1 * 0.4 * "x");
    "phi" := "phi" + "w0c_3_26_2" * SIN(2 * 0.4 * "x") + "w0d_3_26_2" * COS(2 * 0.4 * "x");
    "phi" := "phi" + "w0c_3_26_3" * SIN(3 * 0.4 * "x") + "w0d_3_26_3" * COS(3 * 0.4 * "x");
    "phi" := "phi" + "w0c_3_26_4" * SIN(4 * 0.4 * "x") + "w0d_3_26_4" * COS(4 * 0.4 * "x");
    "phi" := "phi" + "w0c_3_26_5" * SIN(5 * 0.4 * "x") + "w0d_3_26_5" * COS(5 * 0.4 * "x");
    "phi" := "phi" + "w0c_3_26_6" * SIN(6 * 0.4 * "x") + "w0d_3_26_6" * COS(6 * 0.4 * "x");
    "acc" := "acc" + "phi";
    "x" := "feat_27";
    "phi" := "w0b_3_27" * "x" / (1.0 + EXP(-"x"));
    "phi" := "phi" + "w0c_3_27_1" * SIN(1 * 0.4 * "x") + "w0d_3_27_1" * COS(1 * 0.4 * "x");
    "phi" := "phi" + "w0c_3_27_2" * SIN(2 * 0.4 * "x") + "w0d_3_27_2" * COS(2 * 0.4 * "x");
    "phi" := "phi" + "w0c_3_27_3" * SIN(3 * 0.4 * "x") + "w0d_3_27_3" * COS(3 * 0.4 * "x");
    "phi" := "phi" + "w0c_3_27_4" * SIN(4 * 0.4 * "x") + "w0d_3_27_4" * COS(4 * 0.4 * "x");
    "phi" := "phi" + "w0c_3_27_5" * SIN(5 * 0.4 * "x") + "w0d_3_27_5" * COS(5 * 0.4 * "x");
    "phi" := "phi" + "w0c_3_27_6" * SIN(6 * 0.4 * "x") + "w0d_3_27_6" * COS(6 * 0.4 * "x");
    "acc" := "acc" + "phi";
    "x" := "feat_28";
    "phi" := "w0b_3_28" * "x" / (1.0 + EXP(-"x"));
    "phi" := "phi" + "w0c_3_28_1" * SIN(1 * 0.4 * "x") + "w0d_3_28_1" * COS(1 * 0.4 * "x");
    "phi" := "phi" + "w0c_3_28_2" * SIN(2 * 0.4 * "x") + "w0d_3_28_2" * COS(2 * 0.4 * "x");
    "phi" := "phi" + "w0c_3_28_3" * SIN(3 * 0.4 * "x") + "w0d_3_28_3" * COS(3 * 0.4 * "x");
    "phi" := "phi" + "w0c_3_28_4" * SIN(4 * 0.4 * "x") + "w0d_3_28_4" * COS(4 * 0.4 * "x");
    "phi" := "phi" + "w0c_3_28_5" * SIN(5 * 0.4 * "x") + "w0d_3_28_5" * COS(5 * 0.4 * "x");
    "phi" := "phi" + "w0c_3_28_6" * SIN(6 * 0.4 * "x") + "w0d_3_28_6" * COS(6 * 0.4 * "x");
    "acc" := "acc" + "phi";
    "h1_3" := "acc" + "b0_3";
    "acc" := 0.0;
    "x" := "feat_1";
    "phi" := "w0b_4_1" * "x" / (1.0 + EXP(-"x"));
    "phi" := "phi" + "w0c_4_1_1" * SIN(1 * 0.4 * "x") + "w0d_4_1_1" * COS(1 * 0.4 * "x");
    "phi" := "phi" + "w0c_4_1_2" * SIN(2 * 0.4 * "x") + "w0d_4_1_2" * COS(2 * 0.4 * "x");
    "phi" := "phi" + "w0c_4_1_3" * SIN(3 * 0.4 * "x") + "w0d_4_1_3" * COS(3 * 0.4 * "x");
    "phi" := "phi" + "w0c_4_1_4" * SIN(4 * 0.4 * "x") + "w0d_4_1_4" * COS(4 * 0.4 * "x");
    "phi" := "phi" + "w0c_4_1_5" * SIN(5 * 0.4 * "x") + "w0d_4_1_5" * COS(5 * 0.4 * "x");
    "phi" := "phi" + "w0c_4_1_6" * SIN(6 * 0.4 * "x") + "w0d_4_1_6" * COS(6 * 0.4 * "x");
    "acc" := "acc" + "phi";
    "x" := "feat_2";
    "phi" := "w0b_4_2" * "x" / (1.0 + EXP(-"x"));
    "phi" := "phi" + "w0c_4_2_1" * SIN(1 * 0.4 * "x") + "w0d_4_2_1" * COS(1 * 0.4 * "x");
    "phi" := "phi" + "w0c_4_2_2" * SIN(2 * 0.4 * "x") + "w0d_4_2_2" * COS(2 * 0.4 * "x");
    "phi" := "phi" + "w0c_4_2_3" * SIN(3 * 0.4 * "x") + "w0d_4_2_3" * COS(3 * 0.4 * "x");
    "phi" := "phi" + "w0c_4_2_4" * SIN(4 * 0.4 * "x") + "w0d_4_2_4" * COS(4 * 0.4 * "x");
    "phi" := "phi" + "w0c_4_2_5" * SIN(5 * 0.4 * "x") + "w0d_4_2_5" * COS(5 * 0.4 * "x");
    "phi" := "phi" + "w0c_4_2_6" * SIN(6 * 0.4 * "x") + "w0d_4_2_6" * COS(6 * 0.4 * "x");
    "acc" := "acc" + "phi";
    "x" := "feat_3";
    "phi" := "w0b_4_3" * "x" / (1.0 + EXP(-"x"));
    "phi" := "phi" + "w0c_4_3_1" * SIN(1 * 0.4 * "x") + "w0d_4_3_1" * COS(1 * 0.4 * "x");
    "phi" := "phi" + "w0c_4_3_2" * SIN(2 * 0.4 * "x") + "w0d_4_3_2" * COS(2 * 0.4 * "x");
    "phi" := "phi" + "w0c_4_3_3" * SIN(3 * 0.4 * "x") + "w0d_4_3_3" * COS(3 * 0.4 * "x");
    "phi" := "phi" + "w0c_4_3_4" * SIN(4 * 0.4 * "x") + "w0d_4_3_4" * COS(4 * 0.4 * "x");
    "phi" := "phi" + "w0c_4_3_5" * SIN(5 * 0.4 * "x") + "w0d_4_3_5" * COS(5 * 0.4 * "x");
    "phi" := "phi" + "w0c_4_3_6" * SIN(6 * 0.4 * "x") + "w0d_4_3_6" * COS(6 * 0.4 * "x");
    "acc" := "acc" + "phi";
    "x" := "feat_4";
    "phi" := "w0b_4_4" * "x" / (1.0 + EXP(-"x"));
    "phi" := "phi" + "w0c_4_4_1" * SIN(1 * 0.4 * "x") + "w0d_4_4_1" * COS(1 * 0.4 * "x");
    "phi" := "phi" + "w0c_4_4_2" * SIN(2 * 0.4 * "x") + "w0d_4_4_2" * COS(2 * 0.4 * "x");
    "phi" := "phi" + "w0c_4_4_3" * SIN(3 * 0.4 * "x") + "w0d_4_4_3" * COS(3 * 0.4 * "x");
    "phi" := "phi" + "w0c_4_4_4" * SIN(4 * 0.4 * "x") + "w0d_4_4_4" * COS(4 * 0.4 * "x");
    "phi" := "phi" + "w0c_4_4_5" * SIN(5 * 0.4 * "x") + "w0d_4_4_5" * COS(5 * 0.4 * "x");
    "phi" := "phi" + "w0c_4_4_6" * SIN(6 * 0.4 * "x") + "w0d_4_4_6" * COS(6 * 0.4 * "x");
    "acc" := "acc" + "phi";
    "x" := "feat_5";
    "phi" := "w0b_4_5" * "x" / (1.0 + EXP(-"x"));
    "phi" := "phi" + "w0c_4_5_1" * SIN(1 * 0.4 * "x") + "w0d_4_5_1" * COS(1 * 0.4 * "x");
    "phi" := "phi" + "w0c_4_5_2" * SIN(2 * 0.4 * "x") + "w0d_4_5_2" * COS(2 * 0.4 * "x");
    "phi" := "phi" + "w0c_4_5_3" * SIN(3 * 0.4 * "x") + "w0d_4_5_3" * COS(3 * 0.4 * "x");
    "phi" := "phi" + "w0c_4_5_4" * SIN(4 * 0.4 * "x") + "w0d_4_5_4" * COS(4 * 0.4 * "x");
    "phi" := "phi" + "w0c_4_5_5" * SIN(5 * 0.4 * "x") + "w0d_4_5_5" * COS(5 * 0.4 * "x");
    "phi" := "phi" + "w0c_4_5_6" * SIN(6 * 0.4 * "x") + "w0d_4_5_6" * COS(6 * 0.4 * "x");
    "acc" := "acc" + "phi";
    "x" := "feat_6";
    "phi" := "w0b_4_6" * "x" / (1.0 + EXP(-"x"));
    "phi" := "phi" + "w0c_4_6_1" * SIN(1 * 0.4 * "x") + "w0d_4_6_1" * COS(1 * 0.4 * "x");
    "phi" := "phi" + "w0c_4_6_2" * SIN(2 * 0.4 * "x") + "w0d_4_6_2" * COS(2 * 0.4 * "x");
    "phi" := "phi" + "w0c_4_6_3" * SIN(3 * 0.4 * "x") + "w0d_4_6_3" * COS(3 * 0.4 * "x");
    "phi" := "phi" + "w0c_4_6_4" * SIN(4 * 0.4 * "x") + "w0d_4_6_4" * COS(4 * 0.4 * "x");
    "phi" := "phi" + "w0c_4_6_5" * SIN(5 * 0.4 * "x") + "w0d_4_6_5" * COS(5 * 0.4 * "x");
    "phi" := "phi" + "w0c_4_6_6" * SIN(6 * 0.4 * "x") + "w0d_4_6_6" * COS(6 * 0.4 * "x");
    "acc" := "acc" + "phi";
    "x" := "feat_7";
    "phi" := "w0b_4_7" * "x" / (1.0 + EXP(-"x"));
    "phi" := "phi" + "w0c_4_7_1" * SIN(1 * 0.4 * "x") + "w0d_4_7_1" * COS(1 * 0.4 * "x");
    "phi" := "phi" + "w0c_4_7_2" * SIN(2 * 0.4 * "x") + "w0d_4_7_2" * COS(2 * 0.4 * "x");
    "phi" := "phi" + "w0c_4_7_3" * SIN(3 * 0.4 * "x") + "w0d_4_7_3" * COS(3 * 0.4 * "x");
    "phi" := "phi" + "w0c_4_7_4" * SIN(4 * 0.4 * "x") + "w0d_4_7_4" * COS(4 * 0.4 * "x");
    "phi" := "phi" + "w0c_4_7_5" * SIN(5 * 0.4 * "x") + "w0d_4_7_5" * COS(5 * 0.4 * "x");
    "phi" := "phi" + "w0c_4_7_6" * SIN(6 * 0.4 * "x") + "w0d_4_7_6" * COS(6 * 0.4 * "x");
    "acc" := "acc" + "phi";
    "x" := "feat_8";
    "phi" := "w0b_4_8" * "x" / (1.0 + EXP(-"x"));
    "phi" := "phi" + "w0c_4_8_1" * SIN(1 * 0.4 * "x") + "w0d_4_8_1" * COS(1 * 0.4 * "x");
    "phi" := "phi" + "w0c_4_8_2" * SIN(2 * 0.4 * "x") + "w0d_4_8_2" * COS(2 * 0.4 * "x");
    "phi" := "phi" + "w0c_4_8_3" * SIN(3 * 0.4 * "x") + "w0d_4_8_3" * COS(3 * 0.4 * "x");
    "phi" := "phi" + "w0c_4_8_4" * SIN(4 * 0.4 * "x") + "w0d_4_8_4" * COS(4 * 0.4 * "x");
    "phi" := "phi" + "w0c_4_8_5" * SIN(5 * 0.4 * "x") + "w0d_4_8_5" * COS(5 * 0.4 * "x");
    "phi" := "phi" + "w0c_4_8_6" * SIN(6 * 0.4 * "x") + "w0d_4_8_6" * COS(6 * 0.4 * "x");
    "acc" := "acc" + "phi";
    "x" := "feat_9";
    "phi" := "w0b_4_9" * "x" / (1.0 + EXP(-"x"));
    "phi" := "phi" + "w0c_4_9_1" * SIN(1 * 0.4 * "x") + "w0d_4_9_1" * COS(1 * 0.4 * "x");
    "phi" := "phi" + "w0c_4_9_2" * SIN(2 * 0.4 * "x") + "w0d_4_9_2" * COS(2 * 0.4 * "x");
    "phi" := "phi" + "w0c_4_9_3" * SIN(3 * 0.4 * "x") + "w0d_4_9_3" * COS(3 * 0.4 * "x");
    "phi" := "phi" + "w0c_4_9_4" * SIN(4 * 0.4 * "x") + "w0d_4_9_4" * COS(4 * 0.4 * "x");
    "phi" := "phi" + "w0c_4_9_5" * SIN(5 * 0.4 * "x") + "w0d_4_9_5" * COS(5 * 0.4 * "x");
    "phi" := "phi" + "w0c_4_9_6" * SIN(6 * 0.4 * "x") + "w0d_4_9_6" * COS(6 * 0.4 * "x");
    "acc" := "acc" + "phi";
    "x" := "feat_10";
    "phi" := "w0b_4_10" * "x" / (1.0 + EXP(-"x"));
    "phi" := "phi" + "w0c_4_10_1" * SIN(1 * 0.4 * "x") + "w0d_4_10_1" * COS(1 * 0.4 * "x");
    "phi" := "phi" + "w0c_4_10_2" * SIN(2 * 0.4 * "x") + "w0d_4_10_2" * COS(2 * 0.4 * "x");
    "phi" := "phi" + "w0c_4_10_3" * SIN(3 * 0.4 * "x") + "w0d_4_10_3" * COS(3 * 0.4 * "x");
    "phi" := "phi" + "w0c_4_10_4" * SIN(4 * 0.4 * "x") + "w0d_4_10_4" * COS(4 * 0.4 * "x");
    "phi" := "phi" + "w0c_4_10_5" * SIN(5 * 0.4 * "x") + "w0d_4_10_5" * COS(5 * 0.4 * "x");
    "phi" := "phi" + "w0c_4_10_6" * SIN(6 * 0.4 * "x") + "w0d_4_10_6" * COS(6 * 0.4 * "x");
    "acc" := "acc" + "phi";
    "x" := "feat_11";
    "phi" := "w0b_4_11" * "x" / (1.0 + EXP(-"x"));
    "phi" := "phi" + "w0c_4_11_1" * SIN(1 * 0.4 * "x") + "w0d_4_11_1" * COS(1 * 0.4 * "x");
    "phi" := "phi" + "w0c_4_11_2" * SIN(2 * 0.4 * "x") + "w0d_4_11_2" * COS(2 * 0.4 * "x");
    "phi" := "phi" + "w0c_4_11_3" * SIN(3 * 0.4 * "x") + "w0d_4_11_3" * COS(3 * 0.4 * "x");
    "phi" := "phi" + "w0c_4_11_4" * SIN(4 * 0.4 * "x") + "w0d_4_11_4" * COS(4 * 0.4 * "x");
    "phi" := "phi" + "w0c_4_11_5" * SIN(5 * 0.4 * "x") + "w0d_4_11_5" * COS(5 * 0.4 * "x");
    "phi" := "phi" + "w0c_4_11_6" * SIN(6 * 0.4 * "x") + "w0d_4_11_6" * COS(6 * 0.4 * "x");
    "acc" := "acc" + "phi";
    "x" := "feat_12";
    "phi" := "w0b_4_12" * "x" / (1.0 + EXP(-"x"));
    "phi" := "phi" + "w0c_4_12_1" * SIN(1 * 0.4 * "x") + "w0d_4_12_1" * COS(1 * 0.4 * "x");
    "phi" := "phi" + "w0c_4_12_2" * SIN(2 * 0.4 * "x") + "w0d_4_12_2" * COS(2 * 0.4 * "x");
    "phi" := "phi" + "w0c_4_12_3" * SIN(3 * 0.4 * "x") + "w0d_4_12_3" * COS(3 * 0.4 * "x");
    "phi" := "phi" + "w0c_4_12_4" * SIN(4 * 0.4 * "x") + "w0d_4_12_4" * COS(4 * 0.4 * "x");
    "phi" := "phi" + "w0c_4_12_5" * SIN(5 * 0.4 * "x") + "w0d_4_12_5" * COS(5 * 0.4 * "x");
    "phi" := "phi" + "w0c_4_12_6" * SIN(6 * 0.4 * "x") + "w0d_4_12_6" * COS(6 * 0.4 * "x");
    "acc" := "acc" + "phi";
    "x" := "feat_13";
    "phi" := "w0b_4_13" * "x" / (1.0 + EXP(-"x"));
    "phi" := "phi" + "w0c_4_13_1" * SIN(1 * 0.4 * "x") + "w0d_4_13_1" * COS(1 * 0.4 * "x");
    "phi" := "phi" + "w0c_4_13_2" * SIN(2 * 0.4 * "x") + "w0d_4_13_2" * COS(2 * 0.4 * "x");
    "phi" := "phi" + "w0c_4_13_3" * SIN(3 * 0.4 * "x") + "w0d_4_13_3" * COS(3 * 0.4 * "x");
    "phi" := "phi" + "w0c_4_13_4" * SIN(4 * 0.4 * "x") + "w0d_4_13_4" * COS(4 * 0.4 * "x");
    "phi" := "phi" + "w0c_4_13_5" * SIN(5 * 0.4 * "x") + "w0d_4_13_5" * COS(5 * 0.4 * "x");
    "phi" := "phi" + "w0c_4_13_6" * SIN(6 * 0.4 * "x") + "w0d_4_13_6" * COS(6 * 0.4 * "x");
    "acc" := "acc" + "phi";
    "x" := "feat_14";
    "phi" := "w0b_4_14" * "x" / (1.0 + EXP(-"x"));
    "phi" := "phi" + "w0c_4_14_1" * SIN(1 * 0.4 * "x") + "w0d_4_14_1" * COS(1 * 0.4 * "x");
    "phi" := "phi" + "w0c_4_14_2" * SIN(2 * 0.4 * "x") + "w0d_4_14_2" * COS(2 * 0.4 * "x");
    "phi" := "phi" + "w0c_4_14_3" * SIN(3 * 0.4 * "x") + "w0d_4_14_3" * COS(3 * 0.4 * "x");
    "phi" := "phi" + "w0c_4_14_4" * SIN(4 * 0.4 * "x") + "w0d_4_14_4" * COS(4 * 0.4 * "x");
    "phi" := "phi" + "w0c_4_14_5" * SIN(5 * 0.4 * "x") + "w0d_4_14_5" * COS(5 * 0.4 * "x");
    "phi" := "phi" + "w0c_4_14_6" * SIN(6 * 0.4 * "x") + "w0d_4_14_6" * COS(6 * 0.4 * "x");
    "acc" := "acc" + "phi";
    "x" := "feat_15";
    "phi" := "w0b_4_15" * "x" / (1.0 + EXP(-"x"));
    "phi" := "phi" + "w0c_4_15_1" * SIN(1 * 0.4 * "x") + "w0d_4_15_1" * COS(1 * 0.4 * "x");
    "phi" := "phi" + "w0c_4_15_2" * SIN(2 * 0.4 * "x") + "w0d_4_15_2" * COS(2 * 0.4 * "x");
    "phi" := "phi" + "w0c_4_15_3" * SIN(3 * 0.4 * "x") + "w0d_4_15_3" * COS(3 * 0.4 * "x");
    "phi" := "phi" + "w0c_4_15_4" * SIN(4 * 0.4 * "x") + "w0d_4_15_4" * COS(4 * 0.4 * "x");
    "phi" := "phi" + "w0c_4_15_5" * SIN(5 * 0.4 * "x") + "w0d_4_15_5" * COS(5 * 0.4 * "x");
    "phi" := "phi" + "w0c_4_15_6" * SIN(6 * 0.4 * "x") + "w0d_4_15_6" * COS(6 * 0.4 * "x");
    "acc" := "acc" + "phi";
    "x" := "feat_16";
    "phi" := "w0b_4_16" * "x" / (1.0 + EXP(-"x"));
    "phi" := "phi" + "w0c_4_16_1" * SIN(1 * 0.4 * "x") + "w0d_4_16_1" * COS(1 * 0.4 * "x");
    "phi" := "phi" + "w0c_4_16_2" * SIN(2 * 0.4 * "x") + "w0d_4_16_2" * COS(2 * 0.4 * "x");
    "phi" := "phi" + "w0c_4_16_3" * SIN(3 * 0.4 * "x") + "w0d_4_16_3" * COS(3 * 0.4 * "x");
    "phi" := "phi" + "w0c_4_16_4" * SIN(4 * 0.4 * "x") + "w0d_4_16_4" * COS(4 * 0.4 * "x");
    "phi" := "phi" + "w0c_4_16_5" * SIN(5 * 0.4 * "x") + "w0d_4_16_5" * COS(5 * 0.4 * "x");
    "phi" := "phi" + "w0c_4_16_6" * SIN(6 * 0.4 * "x") + "w0d_4_16_6" * COS(6 * 0.4 * "x");
    "acc" := "acc" + "phi";
    "x" := "feat_17";
    "phi" := "w0b_4_17" * "x" / (1.0 + EXP(-"x"));
    "phi" := "phi" + "w0c_4_17_1" * SIN(1 * 0.4 * "x") + "w0d_4_17_1" * COS(1 * 0.4 * "x");
    "phi" := "phi" + "w0c_4_17_2" * SIN(2 * 0.4 * "x") + "w0d_4_17_2" * COS(2 * 0.4 * "x");
    "phi" := "phi" + "w0c_4_17_3" * SIN(3 * 0.4 * "x") + "w0d_4_17_3" * COS(3 * 0.4 * "x");
    "phi" := "phi" + "w0c_4_17_4" * SIN(4 * 0.4 * "x") + "w0d_4_17_4" * COS(4 * 0.4 * "x");
    "phi" := "phi" + "w0c_4_17_5" * SIN(5 * 0.4 * "x") + "w0d_4_17_5" * COS(5 * 0.4 * "x");
    "phi" := "phi" + "w0c_4_17_6" * SIN(6 * 0.4 * "x") + "w0d_4_17_6" * COS(6 * 0.4 * "x");
    "acc" := "acc" + "phi";
    "x" := "feat_18";
    "phi" := "w0b_4_18" * "x" / (1.0 + EXP(-"x"));
    "phi" := "phi" + "w0c_4_18_1" * SIN(1 * 0.4 * "x") + "w0d_4_18_1" * COS(1 * 0.4 * "x");
    "phi" := "phi" + "w0c_4_18_2" * SIN(2 * 0.4 * "x") + "w0d_4_18_2" * COS(2 * 0.4 * "x");
    "phi" := "phi" + "w0c_4_18_3" * SIN(3 * 0.4 * "x") + "w0d_4_18_3" * COS(3 * 0.4 * "x");
    "phi" := "phi" + "w0c_4_18_4" * SIN(4 * 0.4 * "x") + "w0d_4_18_4" * COS(4 * 0.4 * "x");
    "phi" := "phi" + "w0c_4_18_5" * SIN(5 * 0.4 * "x") + "w0d_4_18_5" * COS(5 * 0.4 * "x");
    "phi" := "phi" + "w0c_4_18_6" * SIN(6 * 0.4 * "x") + "w0d_4_18_6" * COS(6 * 0.4 * "x");
    "acc" := "acc" + "phi";
    "x" := "feat_19";
    "phi" := "w0b_4_19" * "x" / (1.0 + EXP(-"x"));
    "phi" := "phi" + "w0c_4_19_1" * SIN(1 * 0.4 * "x") + "w0d_4_19_1" * COS(1 * 0.4 * "x");
    "phi" := "phi" + "w0c_4_19_2" * SIN(2 * 0.4 * "x") + "w0d_4_19_2" * COS(2 * 0.4 * "x");
    "phi" := "phi" + "w0c_4_19_3" * SIN(3 * 0.4 * "x") + "w0d_4_19_3" * COS(3 * 0.4 * "x");
    "phi" := "phi" + "w0c_4_19_4" * SIN(4 * 0.4 * "x") + "w0d_4_19_4" * COS(4 * 0.4 * "x");
    "phi" := "phi" + "w0c_4_19_5" * SIN(5 * 0.4 * "x") + "w0d_4_19_5" * COS(5 * 0.4 * "x");
    "phi" := "phi" + "w0c_4_19_6" * SIN(6 * 0.4 * "x") + "w0d_4_19_6" * COS(6 * 0.4 * "x");
    "acc" := "acc" + "phi";
    "x" := "feat_20";
    "phi" := "w0b_4_20" * "x" / (1.0 + EXP(-"x"));
    "phi" := "phi" + "w0c_4_20_1" * SIN(1 * 0.4 * "x") + "w0d_4_20_1" * COS(1 * 0.4 * "x");
    "phi" := "phi" + "w0c_4_20_2" * SIN(2 * 0.4 * "x") + "w0d_4_20_2" * COS(2 * 0.4 * "x");
    "phi" := "phi" + "w0c_4_20_3" * SIN(3 * 0.4 * "x") + "w0d_4_20_3" * COS(3 * 0.4 * "x");
    "phi" := "phi" + "w0c_4_20_4" * SIN(4 * 0.4 * "x") + "w0d_4_20_4" * COS(4 * 0.4 * "x");
    "phi" := "phi" + "w0c_4_20_5" * SIN(5 * 0.4 * "x") + "w0d_4_20_5" * COS(5 * 0.4 * "x");
    "phi" := "phi" + "w0c_4_20_6" * SIN(6 * 0.4 * "x") + "w0d_4_20_6" * COS(6 * 0.4 * "x");
    "acc" := "acc" + "phi";
    "x" := "feat_21";
    "phi" := "w0b_4_21" * "x" / (1.0 + EXP(-"x"));
    "phi" := "phi" + "w0c_4_21_1" * SIN(1 * 0.4 * "x") + "w0d_4_21_1" * COS(1 * 0.4 * "x");
    "phi" := "phi" + "w0c_4_21_2" * SIN(2 * 0.4 * "x") + "w0d_4_21_2" * COS(2 * 0.4 * "x");
    "phi" := "phi" + "w0c_4_21_3" * SIN(3 * 0.4 * "x") + "w0d_4_21_3" * COS(3 * 0.4 * "x");
    "phi" := "phi" + "w0c_4_21_4" * SIN(4 * 0.4 * "x") + "w0d_4_21_4" * COS(4 * 0.4 * "x");
    "phi" := "phi" + "w0c_4_21_5" * SIN(5 * 0.4 * "x") + "w0d_4_21_5" * COS(5 * 0.4 * "x");
    "phi" := "phi" + "w0c_4_21_6" * SIN(6 * 0.4 * "x") + "w0d_4_21_6" * COS(6 * 0.4 * "x");
    "acc" := "acc" + "phi";
    "x" := "feat_22";
    "phi" := "w0b_4_22" * "x" / (1.0 + EXP(-"x"));
    "phi" := "phi" + "w0c_4_22_1" * SIN(1 * 0.4 * "x") + "w0d_4_22_1" * COS(1 * 0.4 * "x");
    "phi" := "phi" + "w0c_4_22_2" * SIN(2 * 0.4 * "x") + "w0d_4_22_2" * COS(2 * 0.4 * "x");
    "phi" := "phi" + "w0c_4_22_3" * SIN(3 * 0.4 * "x") + "w0d_4_22_3" * COS(3 * 0.4 * "x");
    "phi" := "phi" + "w0c_4_22_4" * SIN(4 * 0.4 * "x") + "w0d_4_22_4" * COS(4 * 0.4 * "x");
    "phi" := "phi" + "w0c_4_22_5" * SIN(5 * 0.4 * "x") + "w0d_4_22_5" * COS(5 * 0.4 * "x");
    "phi" := "phi" + "w0c_4_22_6" * SIN(6 * 0.4 * "x") + "w0d_4_22_6" * COS(6 * 0.4 * "x");
    "acc" := "acc" + "phi";
    "x" := "feat_23";
    "phi" := "w0b_4_23" * "x" / (1.0 + EXP(-"x"));
    "phi" := "phi" + "w0c_4_23_1" * SIN(1 * 0.4 * "x") + "w0d_4_23_1" * COS(1 * 0.4 * "x");
    "phi" := "phi" + "w0c_4_23_2" * SIN(2 * 0.4 * "x") + "w0d_4_23_2" * COS(2 * 0.4 * "x");
    "phi" := "phi" + "w0c_4_23_3" * SIN(3 * 0.4 * "x") + "w0d_4_23_3" * COS(3 * 0.4 * "x");
    "phi" := "phi" + "w0c_4_23_4" * SIN(4 * 0.4 * "x") + "w0d_4_23_4" * COS(4 * 0.4 * "x");
    "phi" := "phi" + "w0c_4_23_5" * SIN(5 * 0.4 * "x") + "w0d_4_23_5" * COS(5 * 0.4 * "x");
    "phi" := "phi" + "w0c_4_23_6" * SIN(6 * 0.4 * "x") + "w0d_4_23_6" * COS(6 * 0.4 * "x");
    "acc" := "acc" + "phi";
    "x" := "feat_24";
    "phi" := "w0b_4_24" * "x" / (1.0 + EXP(-"x"));
    "phi" := "phi" + "w0c_4_24_1" * SIN(1 * 0.4 * "x") + "w0d_4_24_1" * COS(1 * 0.4 * "x");
    "phi" := "phi" + "w0c_4_24_2" * SIN(2 * 0.4 * "x") + "w0d_4_24_2" * COS(2 * 0.4 * "x");
    "phi" := "phi" + "w0c_4_24_3" * SIN(3 * 0.4 * "x") + "w0d_4_24_3" * COS(3 * 0.4 * "x");
    "phi" := "phi" + "w0c_4_24_4" * SIN(4 * 0.4 * "x") + "w0d_4_24_4" * COS(4 * 0.4 * "x");
    "phi" := "phi" + "w0c_4_24_5" * SIN(5 * 0.4 * "x") + "w0d_4_24_5" * COS(5 * 0.4 * "x");
    "phi" := "phi" + "w0c_4_24_6" * SIN(6 * 0.4 * "x") + "w0d_4_24_6" * COS(6 * 0.4 * "x");
    "acc" := "acc" + "phi";
    "x" := "feat_25";
    "phi" := "w0b_4_25" * "x" / (1.0 + EXP(-"x"));
    "phi" := "phi" + "w0c_4_25_1" * SIN(1 * 0.4 * "x") + "w0d_4_25_1" * COS(1 * 0.4 * "x");
    "phi" := "phi" + "w0c_4_25_2" * SIN(2 * 0.4 * "x") + "w0d_4_25_2" * COS(2 * 0.4 * "x");
    "phi" := "phi" + "w0c_4_25_3" * SIN(3 * 0.4 * "x") + "w0d_4_25_3" * COS(3 * 0.4 * "x");
    "phi" := "phi" + "w0c_4_25_4" * SIN(4 * 0.4 * "x") + "w0d_4_25_4" * COS(4 * 0.4 * "x");
    "phi" := "phi" + "w0c_4_25_5" * SIN(5 * 0.4 * "x") + "w0d_4_25_5" * COS(5 * 0.4 * "x");
    "phi" := "phi" + "w0c_4_25_6" * SIN(6 * 0.4 * "x") + "w0d_4_25_6" * COS(6 * 0.4 * "x");
    "acc" := "acc" + "phi";
    "x" := "feat_26";
    "phi" := "w0b_4_26" * "x" / (1.0 + EXP(-"x"));
    "phi" := "phi" + "w0c_4_26_1" * SIN(1 * 0.4 * "x") + "w0d_4_26_1" * COS(1 * 0.4 * "x");
    "phi" := "phi" + "w0c_4_26_2" * SIN(2 * 0.4 * "x") + "w0d_4_26_2" * COS(2 * 0.4 * "x");
    "phi" := "phi" + "w0c_4_26_3" * SIN(3 * 0.4 * "x") + "w0d_4_26_3" * COS(3 * 0.4 * "x");
    "phi" := "phi" + "w0c_4_26_4" * SIN(4 * 0.4 * "x") + "w0d_4_26_4" * COS(4 * 0.4 * "x");
    "phi" := "phi" + "w0c_4_26_5" * SIN(5 * 0.4 * "x") + "w0d_4_26_5" * COS(5 * 0.4 * "x");
    "phi" := "phi" + "w0c_4_26_6" * SIN(6 * 0.4 * "x") + "w0d_4_26_6" * COS(6 * 0.4 * "x");
    "acc" := "acc" + "phi";
    "x" := "feat_27";
    "phi" := "w0b_4_27" * "x" / (1.0 + EXP(-"x"));
    "phi" := "phi" + "w0c_4_27_1" * SIN(1 * 0.4 * "x") + "w0d_4_27_1" * COS(1 * 0.4 * "x");
    "phi" := "phi" + "w0c_4_27_2" * SIN(2 * 0.4 * "x") + "w0d_4_27_2" * COS(2 * 0.4 * "x");
    "phi" := "phi" + "w0c_4_27_3" * SIN(3 * 0.4 * "x") + "w0d_4_27_3" * COS(3 * 0.4 * "x");
    "phi" := "phi" + "w0c_4_27_4" * SIN(4 * 0.4 * "x") + "w0d_4_27_4" * COS(4 * 0.4 * "x");
    "phi" := "phi" + "w0c_4_27_5" * SIN(5 * 0.4 * "x") + "w0d_4_27_5" * COS(5 * 0.4 * "x");
    "phi" := "phi" + "w0c_4_27_6" * SIN(6 * 0.4 * "x") + "w0d_4_27_6" * COS(6 * 0.4 * "x");
    "acc" := "acc" + "phi";
    "x" := "feat_28";
    "phi" := "w0b_4_28" * "x" / (1.0 + EXP(-"x"));
    "phi" := "phi" + "w0c_4_28_1" * SIN(1 * 0.4 * "x") + "w0d_4_28_1" * COS(1 * 0.4 * "x");
    "phi" := "phi" + "w0c_4_28_2" * SIN(2 * 0.4 * "x") + "w0d_4_28_2" * COS(2 * 0.4 * "x");
    "phi" := "phi" + "w0c_4_28_3" * SIN(3 * 0.4 * "x") + "w0d_4_28_3" * COS(3 * 0.4 * "x");
    "phi" := "phi" + "w0c_4_28_4" * SIN(4 * 0.4 * "x") + "w0d_4_28_4" * COS(4 * 0.4 * "x");
    "phi" := "phi" + "w0c_4_28_5" * SIN(5 * 0.4 * "x") + "w0d_4_28_5" * COS(5 * 0.4 * "x");
    "phi" := "phi" + "w0c_4_28_6" * SIN(6 * 0.4 * "x") + "w0d_4_28_6" * COS(6 * 0.4 * "x");
    "acc" := "acc" + "phi";
    "h1_4" := "acc" + "b0_4";
    "acc" := 0.0;
    "x" := "feat_1";
    "phi" := "w0b_5_1" * "x" / (1.0 + EXP(-"x"));
    "phi" := "phi" + "w0c_5_1_1" * SIN(1 * 0.4 * "x") + "w0d_5_1_1" * COS(1 * 0.4 * "x");
    "phi" := "phi" + "w0c_5_1_2" * SIN(2 * 0.4 * "x") + "w0d_5_1_2" * COS(2 * 0.4 * "x");
    "phi" := "phi" + "w0c_5_1_3" * SIN(3 * 0.4 * "x") + "w0d_5_1_3" * COS(3 * 0.4 * "x");
    "phi" := "phi" + "w0c_5_1_4" * SIN(4 * 0.4 * "x") + "w0d_5_1_4" * COS(4 * 0.4 * "x");
    "phi" := "phi" + "w0c_5_1_5" * SIN(5 * 0.4 * "x") + "w0d_5_1_5" * COS(5 * 0.4 * "x");
    "phi" := "phi" + "w0c_5_1_6" * SIN(6 * 0.4 * "x") + "w0d_5_1_6" * COS(6 * 0.4 * "x");
    "acc" := "acc" + "phi";
    "x" := "feat_2";
    "phi" := "w0b_5_2" * "x" / (1.0 + EXP(-"x"));
    "phi" := "phi" + "w0c_5_2_1" * SIN(1 * 0.4 * "x") + "w0d_5_2_1" * COS(1 * 0.4 * "x");
    "phi" := "phi" + "w0c_5_2_2" * SIN(2 * 0.4 * "x") + "w0d_5_2_2" * COS(2 * 0.4 * "x");
    "phi" := "phi" + "w0c_5_2_3" * SIN(3 * 0.4 * "x") + "w0d_5_2_3" * COS(3 * 0.4 * "x");
    "phi" := "phi" + "w0c_5_2_4" * SIN(4 * 0.4 * "x") + "w0d_5_2_4" * COS(4 * 0.4 * "x");
    "phi" := "phi" + "w0c_5_2_5" * SIN(5 * 0.4 * "x") + "w0d_5_2_5" * COS(5 * 0.4 * "x");
    "phi" := "phi" + "w0c_5_2_6" * SIN(6 * 0.4 * "x") + "w0d_5_2_6" * COS(6 * 0.4 * "x");
    "acc" := "acc" + "phi";
    "x" := "feat_3";
    "phi" := "w0b_5_3" * "x" / (1.0 + EXP(-"x"));
    "phi" := "phi" + "w0c_5_3_1" * SIN(1 * 0.4 * "x") + "w0d_5_3_1" * COS(1 * 0.4 * "x");
    "phi" := "phi" + "w0c_5_3_2" * SIN(2 * 0.4 * "x") + "w0d_5_3_2" * COS(2 * 0.4 * "x");
    "phi" := "phi" + "w0c_5_3_3" * SIN(3 * 0.4 * "x") + "w0d_5_3_3" * COS(3 * 0.4 * "x");
    "phi" := "phi" + "w0c_5_3_4" * SIN(4 * 0.4 * "x") + "w0d_5_3_4" * COS(4 * 0.4 * "x");
    "phi" := "phi" + "w0c_5_3_5" * SIN(5 * 0.4 * "x") + "w0d_5_3_5" * COS(5 * 0.4 * "x");
    "phi" := "phi" + "w0c_5_3_6" * SIN(6 * 0.4 * "x") + "w0d_5_3_6" * COS(6 * 0.4 * "x");
    "acc" := "acc" + "phi";
    "x" := "feat_4";
    "phi" := "w0b_5_4" * "x" / (1.0 + EXP(-"x"));
    "phi" := "phi" + "w0c_5_4_1" * SIN(1 * 0.4 * "x") + "w0d_5_4_1" * COS(1 * 0.4 * "x");
    "phi" := "phi" + "w0c_5_4_2" * SIN(2 * 0.4 * "x") + "w0d_5_4_2" * COS(2 * 0.4 * "x");
    "phi" := "phi" + "w0c_5_4_3" * SIN(3 * 0.4 * "x") + "w0d_5_4_3" * COS(3 * 0.4 * "x");
    "phi" := "phi" + "w0c_5_4_4" * SIN(4 * 0.4 * "x") + "w0d_5_4_4" * COS(4 * 0.4 * "x");
    "phi" := "phi" + "w0c_5_4_5" * SIN(5 * 0.4 * "x") + "w0d_5_4_5" * COS(5 * 0.4 * "x");
    "phi" := "phi" + "w0c_5_4_6" * SIN(6 * 0.4 * "x") + "w0d_5_4_6" * COS(6 * 0.4 * "x");
    "acc" := "acc" + "phi";
    "x" := "feat_5";
    "phi" := "w0b_5_5" * "x" / (1.0 + EXP(-"x"));
    "phi" := "phi" + "w0c_5_5_1" * SIN(1 * 0.4 * "x") + "w0d_5_5_1" * COS(1 * 0.4 * "x");
    "phi" := "phi" + "w0c_5_5_2" * SIN(2 * 0.4 * "x") + "w0d_5_5_2" * COS(2 * 0.4 * "x");
    "phi" := "phi" + "w0c_5_5_3" * SIN(3 * 0.4 * "x") + "w0d_5_5_3" * COS(3 * 0.4 * "x");
    "phi" := "phi" + "w0c_5_5_4" * SIN(4 * 0.4 * "x") + "w0d_5_5_4" * COS(4 * 0.4 * "x");
    "phi" := "phi" + "w0c_5_5_5" * SIN(5 * 0.4 * "x") + "w0d_5_5_5" * COS(5 * 0.4 * "x");
    "phi" := "phi" + "w0c_5_5_6" * SIN(6 * 0.4 * "x") + "w0d_5_5_6" * COS(6 * 0.4 * "x");
    "acc" := "acc" + "phi";
    "x" := "feat_6";
    "phi" := "w0b_5_6" * "x" / (1.0 + EXP(-"x"));
    "phi" := "phi" + "w0c_5_6_1" * SIN(1 * 0.4 * "x") + "w0d_5_6_1" * COS(1 * 0.4 * "x");
    "phi" := "phi" + "w0c_5_6_2" * SIN(2 * 0.4 * "x") + "w0d_5_6_2" * COS(2 * 0.4 * "x");
    "phi" := "phi" + "w0c_5_6_3" * SIN(3 * 0.4 * "x") + "w0d_5_6_3" * COS(3 * 0.4 * "x");
    "phi" := "phi" + "w0c_5_6_4" * SIN(4 * 0.4 * "x") + "w0d_5_6_4" * COS(4 * 0.4 * "x");
    "phi" := "phi" + "w0c_5_6_5" * SIN(5 * 0.4 * "x") + "w0d_5_6_5" * COS(5 * 0.4 * "x");
    "phi" := "phi" + "w0c_5_6_6" * SIN(6 * 0.4 * "x") + "w0d_5_6_6" * COS(6 * 0.4 * "x");
    "acc" := "acc" + "phi";
    "x" := "feat_7";
    "phi" := "w0b_5_7" * "x" / (1.0 + EXP(-"x"));
    "phi" := "phi" + "w0c_5_7_1" * SIN(1 * 0.4 * "x") + "w0d_5_7_1" * COS(1 * 0.4 * "x");
    "phi" := "phi" + "w0c_5_7_2" * SIN(2 * 0.4 * "x") + "w0d_5_7_2" * COS(2 * 0.4 * "x");
    "phi" := "phi" + "w0c_5_7_3" * SIN(3 * 0.4 * "x") + "w0d_5_7_3" * COS(3 * 0.4 * "x");
    "phi" := "phi" + "w0c_5_7_4" * SIN(4 * 0.4 * "x") + "w0d_5_7_4" * COS(4 * 0.4 * "x");
    "phi" := "phi" + "w0c_5_7_5" * SIN(5 * 0.4 * "x") + "w0d_5_7_5" * COS(5 * 0.4 * "x");
    "phi" := "phi" + "w0c_5_7_6" * SIN(6 * 0.4 * "x") + "w0d_5_7_6" * COS(6 * 0.4 * "x");
    "acc" := "acc" + "phi";
    "x" := "feat_8";
    "phi" := "w0b_5_8" * "x" / (1.0 + EXP(-"x"));
    "phi" := "phi" + "w0c_5_8_1" * SIN(1 * 0.4 * "x") + "w0d_5_8_1" * COS(1 * 0.4 * "x");
    "phi" := "phi" + "w0c_5_8_2" * SIN(2 * 0.4 * "x") + "w0d_5_8_2" * COS(2 * 0.4 * "x");
    "phi" := "phi" + "w0c_5_8_3" * SIN(3 * 0.4 * "x") + "w0d_5_8_3" * COS(3 * 0.4 * "x");
    "phi" := "phi" + "w0c_5_8_4" * SIN(4 * 0.4 * "x") + "w0d_5_8_4" * COS(4 * 0.4 * "x");
    "phi" := "phi" + "w0c_5_8_5" * SIN(5 * 0.4 * "x") + "w0d_5_8_5" * COS(5 * 0.4 * "x");
    "phi" := "phi" + "w0c_5_8_6" * SIN(6 * 0.4 * "x") + "w0d_5_8_6" * COS(6 * 0.4 * "x");
    "acc" := "acc" + "phi";
    "x" := "feat_9";
    "phi" := "w0b_5_9" * "x" / (1.0 + EXP(-"x"));
    "phi" := "phi" + "w0c_5_9_1" * SIN(1 * 0.4 * "x") + "w0d_5_9_1" * COS(1 * 0.4 * "x");
    "phi" := "phi" + "w0c_5_9_2" * SIN(2 * 0.4 * "x") + "w0d_5_9_2" * COS(2 * 0.4 * "x");
    "phi" := "phi" + "w0c_5_9_3" * SIN(3 * 0.4 * "x") + "w0d_5_9_3" * COS(3 * 0.4 * "x");
    "phi" := "phi" + "w0c_5_9_4" * SIN(4 * 0.4 * "x") + "w0d_5_9_4" * COS(4 * 0.4 * "x");
    "phi" := "phi" + "w0c_5_9_5" * SIN(5 * 0.4 * "x") + "w0d_5_9_5" * COS(5 * 0.4 * "x");
    "phi" := "phi" + "w0c_5_9_6" * SIN(6 * 0.4 * "x") + "w0d_5_9_6" * COS(6 * 0.4 * "x");
    "acc" := "acc" + "phi";
    "x" := "feat_10";
    "phi" := "w0b_5_10" * "x" / (1.0 + EXP(-"x"));
    "phi" := "phi" + "w0c_5_10_1" * SIN(1 * 0.4 * "x") + "w0d_5_10_1" * COS(1 * 0.4 * "x");
    "phi" := "phi" + "w0c_5_10_2" * SIN(2 * 0.4 * "x") + "w0d_5_10_2" * COS(2 * 0.4 * "x");
    "phi" := "phi" + "w0c_5_10_3" * SIN(3 * 0.4 * "x") + "w0d_5_10_3" * COS(3 * 0.4 * "x");
    "phi" := "phi" + "w0c_5_10_4" * SIN(4 * 0.4 * "x") + "w0d_5_10_4" * COS(4 * 0.4 * "x");
    "phi" := "phi" + "w0c_5_10_5" * SIN(5 * 0.4 * "x") + "w0d_5_10_5" * COS(5 * 0.4 * "x");
    "phi" := "phi" + "w0c_5_10_6" * SIN(6 * 0.4 * "x") + "w0d_5_10_6" * COS(6 * 0.4 * "x");
    "acc" := "acc" + "phi";
    "x" := "feat_11";
    "phi" := "w0b_5_11" * "x" / (1.0 + EXP(-"x"));
    "phi" := "phi" + "w0c_5_11_1" * SIN(1 * 0.4 * "x") + "w0d_5_11_1" * COS(1 * 0.4 * "x");
    "phi" := "phi" + "w0c_5_11_2" * SIN(2 * 0.4 * "x") + "w0d_5_11_2" * COS(2 * 0.4 * "x");
    "phi" := "phi" + "w0c_5_11_3" * SIN(3 * 0.4 * "x") + "w0d_5_11_3" * COS(3 * 0.4 * "x");
    "phi" := "phi" + "w0c_5_11_4" * SIN(4 * 0.4 * "x") + "w0d_5_11_4" * COS(4 * 0.4 * "x");
    "phi" := "phi" + "w0c_5_11_5" * SIN(5 * 0.4 * "x") + "w0d_5_11_5" * COS(5 * 0.4 * "x");
    "phi" := "phi" + "w0c_5_11_6" * SIN(6 * 0.4 * "x") + "w0d_5_11_6" * COS(6 * 0.4 * "x");
    "acc" := "acc" + "phi";
    "x" := "feat_12";
    "phi" := "w0b_5_12" * "x" / (1.0 + EXP(-"x"));
    "phi" := "phi" + "w0c_5_12_1" * SIN(1 * 0.4 * "x") + "w0d_5_12_1" * COS(1 * 0.4 * "x");
    "phi" := "phi" + "w0c_5_12_2" * SIN(2 * 0.4 * "x") + "w0d_5_12_2" * COS(2 * 0.4 * "x");
    "phi" := "phi" + "w0c_5_12_3" * SIN(3 * 0.4 * "x") + "w0d_5_12_3" * COS(3 * 0.4 * "x");
    "phi" := "phi" + "w0c_5_12_4" * SIN(4 * 0.4 * "x") + "w0d_5_12_4" * COS(4 * 0.4 * "x");
    "phi" := "phi" + "w0c_5_12_5" * SIN(5 * 0.4 * "x") + "w0d_5_12_5" * COS(5 * 0.4 * "x");
    "phi" := "phi" + "w0c_5_12_6" * SIN(6 * 0.4 * "x") + "w0d_5_12_6" * COS(6 * 0.4 * "x");
    "acc" := "acc" + "phi";
    "x" := "feat_13";
    "phi" := "w0b_5_13" * "x" / (1.0 + EXP(-"x"));
    "phi" := "phi" + "w0c_5_13_1" * SIN(1 * 0.4 * "x") + "w0d_5_13_1" * COS(1 * 0.4 * "x");
    "phi" := "phi" + "w0c_5_13_2" * SIN(2 * 0.4 * "x") + "w0d_5_13_2" * COS(2 * 0.4 * "x");
    "phi" := "phi" + "w0c_5_13_3" * SIN(3 * 0.4 * "x") + "w0d_5_13_3" * COS(3 * 0.4 * "x");
    "phi" := "phi" + "w0c_5_13_4" * SIN(4 * 0.4 * "x") + "w0d_5_13_4" * COS(4 * 0.4 * "x");
    "phi" := "phi" + "w0c_5_13_5" * SIN(5 * 0.4 * "x") + "w0d_5_13_5" * COS(5 * 0.4 * "x");
    "phi" := "phi" + "w0c_5_13_6" * SIN(6 * 0.4 * "x") + "w0d_5_13_6" * COS(6 * 0.4 * "x");
    "acc" := "acc" + "phi";
    "x" := "feat_14";
    "phi" := "w0b_5_14" * "x" / (1.0 + EXP(-"x"));
    "phi" := "phi" + "w0c_5_14_1" * SIN(1 * 0.4 * "x") + "w0d_5_14_1" * COS(1 * 0.4 * "x");
    "phi" := "phi" + "w0c_5_14_2" * SIN(2 * 0.4 * "x") + "w0d_5_14_2" * COS(2 * 0.4 * "x");
    "phi" := "phi" + "w0c_5_14_3" * SIN(3 * 0.4 * "x") + "w0d_5_14_3" * COS(3 * 0.4 * "x");
    "phi" := "phi" + "w0c_5_14_4" * SIN(4 * 0.4 * "x") + "w0d_5_14_4" * COS(4 * 0.4 * "x");
    "phi" := "phi" + "w0c_5_14_5" * SIN(5 * 0.4 * "x") + "w0d_5_14_5" * COS(5 * 0.4 * "x");
    "phi" := "phi" + "w0c_5_14_6" * SIN(6 * 0.4 * "x") + "w0d_5_14_6" * COS(6 * 0.4 * "x");
    "acc" := "acc" + "phi";
    "x" := "feat_15";
    "phi" := "w0b_5_15" * "x" / (1.0 + EXP(-"x"));
    "phi" := "phi" + "w0c_5_15_1" * SIN(1 * 0.4 * "x") + "w0d_5_15_1" * COS(1 * 0.4 * "x");
    "phi" := "phi" + "w0c_5_15_2" * SIN(2 * 0.4 * "x") + "w0d_5_15_2" * COS(2 * 0.4 * "x");
    "phi" := "phi" + "w0c_5_15_3" * SIN(3 * 0.4 * "x") + "w0d_5_15_3" * COS(3 * 0.4 * "x");
    "phi" := "phi" + "w0c_5_15_4" * SIN(4 * 0.4 * "x") + "w0d_5_15_4" * COS(4 * 0.4 * "x");
    "phi" := "phi" + "w0c_5_15_5" * SIN(5 * 0.4 * "x") + "w0d_5_15_5" * COS(5 * 0.4 * "x");
    "phi" := "phi" + "w0c_5_15_6" * SIN(6 * 0.4 * "x") + "w0d_5_15_6" * COS(6 * 0.4 * "x");
    "acc" := "acc" + "phi";
    "x" := "feat_16";
    "phi" := "w0b_5_16" * "x" / (1.0 + EXP(-"x"));
    "phi" := "phi" + "w0c_5_16_1" * SIN(1 * 0.4 * "x") + "w0d_5_16_1" * COS(1 * 0.4 * "x");
    "phi" := "phi" + "w0c_5_16_2" * SIN(2 * 0.4 * "x") + "w0d_5_16_2" * COS(2 * 0.4 * "x");
    "phi" := "phi" + "w0c_5_16_3" * SIN(3 * 0.4 * "x") + "w0d_5_16_3" * COS(3 * 0.4 * "x");
    "phi" := "phi" + "w0c_5_16_4" * SIN(4 * 0.4 * "x") + "w0d_5_16_4" * COS(4 * 0.4 * "x");
    "phi" := "phi" + "w0c_5_16_5" * SIN(5 * 0.4 * "x") + "w0d_5_16_5" * COS(5 * 0.4 * "x");
    "phi" := "phi" + "w0c_5_16_6" * SIN(6 * 0.4 * "x") + "w0d_5_16_6" * COS(6 * 0.4 * "x");
    "acc" := "acc" + "phi";
    "x" := "feat_17";
    "phi" := "w0b_5_17" * "x" / (1.0 + EXP(-"x"));
    "phi" := "phi" + "w0c_5_17_1" * SIN(1 * 0.4 * "x") + "w0d_5_17_1" * COS(1 * 0.4 * "x");
    "phi" := "phi" + "w0c_5_17_2" * SIN(2 * 0.4 * "x") + "w0d_5_17_2" * COS(2 * 0.4 * "x");
    "phi" := "phi" + "w0c_5_17_3" * SIN(3 * 0.4 * "x") + "w0d_5_17_3" * COS(3 * 0.4 * "x");
    "phi" := "phi" + "w0c_5_17_4" * SIN(4 * 0.4 * "x") + "w0d_5_17_4" * COS(4 * 0.4 * "x");
    "phi" := "phi" + "w0c_5_17_5" * SIN(5 * 0.4 * "x") + "w0d_5_17_5" * COS(5 * 0.4 * "x");
    "phi" := "phi" + "w0c_5_17_6" * SIN(6 * 0.4 * "x") + "w0d_5_17_6" * COS(6 * 0.4 * "x");
    "acc" := "acc" + "phi";
    "x" := "feat_18";
    "phi" := "w0b_5_18" * "x" / (1.0 + EXP(-"x"));
    "phi" := "phi" + "w0c_5_18_1" * SIN(1 * 0.4 * "x") + "w0d_5_18_1" * COS(1 * 0.4 * "x");
    "phi" := "phi" + "w0c_5_18_2" * SIN(2 * 0.4 * "x") + "w0d_5_18_2" * COS(2 * 0.4 * "x");
    "phi" := "phi" + "w0c_5_18_3" * SIN(3 * 0.4 * "x") + "w0d_5_18_3" * COS(3 * 0.4 * "x");
    "phi" := "phi" + "w0c_5_18_4" * SIN(4 * 0.4 * "x") + "w0d_5_18_4" * COS(4 * 0.4 * "x");
    "phi" := "phi" + "w0c_5_18_5" * SIN(5 * 0.4 * "x") + "w0d_5_18_5" * COS(5 * 0.4 * "x");
    "phi" := "phi" + "w0c_5_18_6" * SIN(6 * 0.4 * "x") + "w0d_5_18_6" * COS(6 * 0.4 * "x");
    "acc" := "acc" + "phi";
    "x" := "feat_19";
    "phi" := "w0b_5_19" * "x" / (1.0 + EXP(-"x"));
    "phi" := "phi" + "w0c_5_19_1" * SIN(1 * 0.4 * "x") + "w0d_5_19_1" * COS(1 * 0.4 * "x");
    "phi" := "phi" + "w0c_5_19_2" * SIN(2 * 0.4 * "x") + "w0d_5_19_2" * COS(2 * 0.4 * "x");
    "phi" := "phi" + "w0c_5_19_3" * SIN(3 * 0.4 * "x") + "w0d_5_19_3" * COS(3 * 0.4 * "x");
    "phi" := "phi" + "w0c_5_19_4" * SIN(4 * 0.4 * "x") + "w0d_5_19_4" * COS(4 * 0.4 * "x");
    "phi" := "phi" + "w0c_5_19_5" * SIN(5 * 0.4 * "x") + "w0d_5_19_5" * COS(5 * 0.4 * "x");
    "phi" := "phi" + "w0c_5_19_6" * SIN(6 * 0.4 * "x") + "w0d_5_19_6" * COS(6 * 0.4 * "x");
    "acc" := "acc" + "phi";
    "x" := "feat_20";
    "phi" := "w0b_5_20" * "x" / (1.0 + EXP(-"x"));
    "phi" := "phi" + "w0c_5_20_1" * SIN(1 * 0.4 * "x") + "w0d_5_20_1" * COS(1 * 0.4 * "x");
    "phi" := "phi" + "w0c_5_20_2" * SIN(2 * 0.4 * "x") + "w0d_5_20_2" * COS(2 * 0.4 * "x");
    "phi" := "phi" + "w0c_5_20_3" * SIN(3 * 0.4 * "x") + "w0d_5_20_3" * COS(3 * 0.4 * "x");
    "phi" := "phi" + "w0c_5_20_4" * SIN(4 * 0.4 * "x") + "w0d_5_20_4" * COS(4 * 0.4 * "x");
    "phi" := "phi" + "w0c_5_20_5" * SIN(5 * 0.4 * "x") + "w0d_5_20_5" * COS(5 * 0.4 * "x");
    "phi" := "phi" + "w0c_5_20_6" * SIN(6 * 0.4 * "x") + "w0d_5_20_6" * COS(6 * 0.4 * "x");
    "acc" := "acc" + "phi";
    "x" := "feat_21";
    "phi" := "w0b_5_21" * "x" / (1.0 + EXP(-"x"));
    "phi" := "phi" + "w0c_5_21_1" * SIN(1 * 0.4 * "x") + "w0d_5_21_1" * COS(1 * 0.4 * "x");
    "phi" := "phi" + "w0c_5_21_2" * SIN(2 * 0.4 * "x") + "w0d_5_21_2" * COS(2 * 0.4 * "x");
    "phi" := "phi" + "w0c_5_21_3" * SIN(3 * 0.4 * "x") + "w0d_5_21_3" * COS(3 * 0.4 * "x");
    "phi" := "phi" + "w0c_5_21_4" * SIN(4 * 0.4 * "x") + "w0d_5_21_4" * COS(4 * 0.4 * "x");
    "phi" := "phi" + "w0c_5_21_5" * SIN(5 * 0.4 * "x") + "w0d_5_21_5" * COS(5 * 0.4 * "x");
    "phi" := "phi" + "w0c_5_21_6" * SIN(6 * 0.4 * "x") + "w0d_5_21_6" * COS(6 * 0.4 * "x");
    "acc" := "acc" + "phi";
    "x" := "feat_22";
    "phi" := "w0b_5_22" * "x" / (1.0 + EXP(-"x"));
    "phi" := "phi" + "w0c_5_22_1" * SIN(1 * 0.4 * "x") + "w0d_5_22_1" * COS(1 * 0.4 * "x");
    "phi" := "phi" + "w0c_5_22_2" * SIN(2 * 0.4 * "x") + "w0d_5_22_2" * COS(2 * 0.4 * "x");
    "phi" := "phi" + "w0c_5_22_3" * SIN(3 * 0.4 * "x") + "w0d_5_22_3" * COS(3 * 0.4 * "x");
    "phi" := "phi" + "w0c_5_22_4" * SIN(4 * 0.4 * "x") + "w0d_5_22_4" * COS(4 * 0.4 * "x");
    "phi" := "phi" + "w0c_5_22_5" * SIN(5 * 0.4 * "x") + "w0d_5_22_5" * COS(5 * 0.4 * "x");
    "phi" := "phi" + "w0c_5_22_6" * SIN(6 * 0.4 * "x") + "w0d_5_22_6" * COS(6 * 0.4 * "x");
    "acc" := "acc" + "phi";
    "x" := "feat_23";
    "phi" := "w0b_5_23" * "x" / (1.0 + EXP(-"x"));
    "phi" := "phi" + "w0c_5_23_1" * SIN(1 * 0.4 * "x") + "w0d_5_23_1" * COS(1 * 0.4 * "x");
    "phi" := "phi" + "w0c_5_23_2" * SIN(2 * 0.4 * "x") + "w0d_5_23_2" * COS(2 * 0.4 * "x");
    "phi" := "phi" + "w0c_5_23_3" * SIN(3 * 0.4 * "x") + "w0d_5_23_3" * COS(3 * 0.4 * "x");
    "phi" := "phi" + "w0c_5_23_4" * SIN(4 * 0.4 * "x") + "w0d_5_23_4" * COS(4 * 0.4 * "x");
    "phi" := "phi" + "w0c_5_23_5" * SIN(5 * 0.4 * "x") + "w0d_5_23_5" * COS(5 * 0.4 * "x");
    "phi" := "phi" + "w0c_5_23_6" * SIN(6 * 0.4 * "x") + "w0d_5_23_6" * COS(6 * 0.4 * "x");
    "acc" := "acc" + "phi";
    "x" := "feat_24";
    "phi" := "w0b_5_24" * "x" / (1.0 + EXP(-"x"));
    "phi" := "phi" + "w0c_5_24_1" * SIN(1 * 0.4 * "x") + "w0d_5_24_1" * COS(1 * 0.4 * "x");
    "phi" := "phi" + "w0c_5_24_2" * SIN(2 * 0.4 * "x") + "w0d_5_24_2" * COS(2 * 0.4 * "x");
    "phi" := "phi" + "w0c_5_24_3" * SIN(3 * 0.4 * "x") + "w0d_5_24_3" * COS(3 * 0.4 * "x");
    "phi" := "phi" + "w0c_5_24_4" * SIN(4 * 0.4 * "x") + "w0d_5_24_4" * COS(4 * 0.4 * "x");
    "phi" := "phi" + "w0c_5_24_5" * SIN(5 * 0.4 * "x") + "w0d_5_24_5" * COS(5 * 0.4 * "x");
    "phi" := "phi" + "w0c_5_24_6" * SIN(6 * 0.4 * "x") + "w0d_5_24_6" * COS(6 * 0.4 * "x");
    "acc" := "acc" + "phi";
    "x" := "feat_25";
    "phi" := "w0b_5_25" * "x" / (1.0 + EXP(-"x"));
    "phi" := "phi" + "w0c_5_25_1" * SIN(1 * 0.4 * "x") + "w0d_5_25_1" * COS(1 * 0.4 * "x");
    "phi" := "phi" + "w0c_5_25_2" * SIN(2 * 0.4 * "x") + "w0d_5_25_2" * COS(2 * 0.4 * "x");
    "phi" := "phi" + "w0c_5_25_3" * SIN(3 * 0.4 * "x") + "w0d_5_25_3" * COS(3 * 0.4 * "x");
    "phi" := "phi" + "w0c_5_25_4" * SIN(4 * 0.4 * "x") + "w0d_5_25_4" * COS(4 * 0.4 * "x");
    "phi" := "phi" + "w0c_5_25_5" * SIN(5 * 0.4 * "x") + "w0d_5_25_5" * COS(5 * 0.4 * "x");
    "phi" := "phi" + "w0c_5_25_6" * SIN(6 * 0.4 * "x") + "w0d_5_25_6" * COS(6 * 0.4 * "x");
    "acc" := "acc" + "phi";
    "x" := "feat_26";
    "phi" := "w0b_5_26" * "x" / (1.0 + EXP(-"x"));
    "phi" := "phi" + "w0c_5_26_1" * SIN(1 * 0.4 * "x") + "w0d_5_26_1" * COS(1 * 0.4 * "x");
    "phi" := "phi" + "w0c_5_26_2" * SIN(2 * 0.4 * "x") + "w0d_5_26_2" * COS(2 * 0.4 * "x");
    "phi" := "phi" + "w0c_5_26_3" * SIN(3 * 0.4 * "x") + "w0d_5_26_3" * COS(3 * 0.4 * "x");
    "phi" := "phi" + "w0c_5_26_4" * SIN(4 * 0.4 * "x") + "w0d_5_26_4" * COS(4 * 0.4 * "x");
    "phi" := "phi" + "w0c_5_26_5" * SIN(5 * 0.4 * "x") + "w0d_5_26_5" * COS(5 * 0.4 * "x");
    "phi" := "phi" + "w0c_5_26_6" * SIN(6 * 0.4 * "x") + "w0d_5_26_6" * COS(6 * 0.4 * "x");
    "acc" := "acc" + "phi";
    "x" := "feat_27";
    "phi" := "w0b_5_27" * "x" / (1.0 + EXP(-"x"));
    "phi" := "phi" + "w0c_5_27_1" * SIN(1 * 0.4 * "x") + "w0d_5_27_1" * COS(1 * 0.4 * "x");
    "phi" := "phi" + "w0c_5_27_2" * SIN(2 * 0.4 * "x") + "w0d_5_27_2" * COS(2 * 0.4 * "x");
    "phi" := "phi" + "w0c_5_27_3" * SIN(3 * 0.4 * "x") + "w0d_5_27_3" * COS(3 * 0.4 * "x");
    "phi" := "phi" + "w0c_5_27_4" * SIN(4 * 0.4 * "x") + "w0d_5_27_4" * COS(4 * 0.4 * "x");
    "phi" := "phi" + "w0c_5_27_5" * SIN(5 * 0.4 * "x") + "w0d_5_27_5" * COS(5 * 0.4 * "x");
    "phi" := "phi" + "w0c_5_27_6" * SIN(6 * 0.4 * "x") + "w0d_5_27_6" * COS(6 * 0.4 * "x");
    "acc" := "acc" + "phi";
    "x" := "feat_28";
    "phi" := "w0b_5_28" * "x" / (1.0 + EXP(-"x"));
    "phi" := "phi" + "w0c_5_28_1" * SIN(1 * 0.4 * "x") + "w0d_5_28_1" * COS(1 * 0.4 * "x");
    "phi" := "phi" + "w0c_5_28_2" * SIN(2 * 0.4 * "x") + "w0d_5_28_2" * COS(2 * 0.4 * "x");
    "phi" := "phi" + "w0c_5_28_3" * SIN(3 * 0.4 * "x") + "w0d_5_28_3" * COS(3 * 0.4 * "x");
    "phi" := "phi" + "w0c_5_28_4" * SIN(4 * 0.4 * "x") + "w0d_5_28_4" * COS(4 * 0.4 * "x");
    "phi" := "phi" + "w0c_5_28_5" * SIN(5 * 0.4 * "x") + "w0d_5_28_5" * COS(5 * 0.4 * "x");
    "phi" := "phi" + "w0c_5_28_6" * SIN(6 * 0.4 * "x") + "w0d_5_28_6" * COS(6 * 0.4 * "x");
    "acc" := "acc" + "phi";
    "h1_5" := "acc" + "b0_5";
    "acc" := 0.0;
    "x" := "feat_1";
    "phi" := "w0b_6_1" * "x" / (1.0 + EXP(-"x"));
    "phi" := "phi" + "w0c_6_1_1" * SIN(1 * 0.4 * "x") + "w0d_6_1_1" * COS(1 * 0.4 * "x");
    "phi" := "phi" + "w0c_6_1_2" * SIN(2 * 0.4 * "x") + "w0d_6_1_2" * COS(2 * 0.4 * "x");
    "phi" := "phi" + "w0c_6_1_3" * SIN(3 * 0.4 * "x") + "w0d_6_1_3" * COS(3 * 0.4 * "x");
    "phi" := "phi" + "w0c_6_1_4" * SIN(4 * 0.4 * "x") + "w0d_6_1_4" * COS(4 * 0.4 * "x");
    "phi" := "phi" + "w0c_6_1_5" * SIN(5 * 0.4 * "x") + "w0d_6_1_5" * COS(5 * 0.4 * "x");
    "phi" := "phi" + "w0c_6_1_6" * SIN(6 * 0.4 * "x") + "w0d_6_1_6" * COS(6 * 0.4 * "x");
    "acc" := "acc" + "phi";
    "x" := "feat_2";
    "phi" := "w0b_6_2" * "x" / (1.0 + EXP(-"x"));
    "phi" := "phi" + "w0c_6_2_1" * SIN(1 * 0.4 * "x") + "w0d_6_2_1" * COS(1 * 0.4 * "x");
    "phi" := "phi" + "w0c_6_2_2" * SIN(2 * 0.4 * "x") + "w0d_6_2_2" * COS(2 * 0.4 * "x");
    "phi" := "phi" + "w0c_6_2_3" * SIN(3 * 0.4 * "x") + "w0d_6_2_3" * COS(3 * 0.4 * "x");
    "phi" := "phi" + "w0c_6_2_4" * SIN(4 * 0.4 * "x") + "w0d_6_2_4" * COS(4 * 0.4 * "x");
    "phi" := "phi" + "w0c_6_2_5" * SIN(5 * 0.4 * "x") + "w0d_6_2_5" * COS(5 * 0.4 * "x");
    "phi" := "phi" + "w0c_6_2_6" * SIN(6 * 0.4 * "x") + "w0d_6_2_6" * COS(6 * 0.4 * "x");
    "acc" := "acc" + "phi";
    "x" := "feat_3";
    "phi" := "w0b_6_3" * "x" / (1.0 + EXP(-"x"));
    "phi" := "phi" + "w0c_6_3_1" * SIN(1 * 0.4 * "x") + "w0d_6_3_1" * COS(1 * 0.4 * "x");
    "phi" := "phi" + "w0c_6_3_2" * SIN(2 * 0.4 * "x") + "w0d_6_3_2" * COS(2 * 0.4 * "x");
    "phi" := "phi" + "w0c_6_3_3" * SIN(3 * 0.4 * "x") + "w0d_6_3_3" * COS(3 * 0.4 * "x");
    "phi" := "phi" + "w0c_6_3_4" * SIN(4 * 0.4 * "x") + "w0d_6_3_4" * COS(4 * 0.4 * "x");
    "phi" := "phi" + "w0c_6_3_5" * SIN(5 * 0.4 * "x") + "w0d_6_3_5" * COS(5 * 0.4 * "x");
    "phi" := "phi" + "w0c_6_3_6" * SIN(6 * 0.4 * "x") + "w0d_6_3_6" * COS(6 * 0.4 * "x");
    "acc" := "acc" + "phi";
    "x" := "feat_4";
    "phi" := "w0b_6_4" * "x" / (1.0 + EXP(-"x"));
    "phi" := "phi" + "w0c_6_4_1" * SIN(1 * 0.4 * "x") + "w0d_6_4_1" * COS(1 * 0.4 * "x");
    "phi" := "phi" + "w0c_6_4_2" * SIN(2 * 0.4 * "x") + "w0d_6_4_2" * COS(2 * 0.4 * "x");
    "phi" := "phi" + "w0c_6_4_3" * SIN(3 * 0.4 * "x") + "w0d_6_4_3" * COS(3 * 0.4 * "x");
    "phi" := "phi" + "w0c_6_4_4" * SIN(4 * 0.4 * "x") + "w0d_6_4_4" * COS(4 * 0.4 * "x");
    "phi" := "phi" + "w0c_6_4_5" * SIN(5 * 0.4 * "x") + "w0d_6_4_5" * COS(5 * 0.4 * "x");
    "phi" := "phi" + "w0c_6_4_6" * SIN(6 * 0.4 * "x") + "w0d_6_4_6" * COS(6 * 0.4 * "x");
    "acc" := "acc" + "phi";
    "x" := "feat_5";
    "phi" := "w0b_6_5" * "x" / (1.0 + EXP(-"x"));
    "phi" := "phi" + "w0c_6_5_1" * SIN(1 * 0.4 * "x") + "w0d_6_5_1" * COS(1 * 0.4 * "x");
    "phi" := "phi" + "w0c_6_5_2" * SIN(2 * 0.4 * "x") + "w0d_6_5_2" * COS(2 * 0.4 * "x");
    "phi" := "phi" + "w0c_6_5_3" * SIN(3 * 0.4 * "x") + "w0d_6_5_3" * COS(3 * 0.4 * "x");
    "phi" := "phi" + "w0c_6_5_4" * SIN(4 * 0.4 * "x") + "w0d_6_5_4" * COS(4 * 0.4 * "x");
    "phi" := "phi" + "w0c_6_5_5" * SIN(5 * 0.4 * "x") + "w0d_6_5_5" * COS(5 * 0.4 * "x");
    "phi" := "phi" + "w0c_6_5_6" * SIN(6 * 0.4 * "x") + "w0d_6_5_6" * COS(6 * 0.4 * "x");
    "acc" := "acc" + "phi";
    "x" := "feat_6";
    "phi" := "w0b_6_6" * "x" / (1.0 + EXP(-"x"));
    "phi" := "phi" + "w0c_6_6_1" * SIN(1 * 0.4 * "x") + "w0d_6_6_1" * COS(1 * 0.4 * "x");
    "phi" := "phi" + "w0c_6_6_2" * SIN(2 * 0.4 * "x") + "w0d_6_6_2" * COS(2 * 0.4 * "x");
    "phi" := "phi" + "w0c_6_6_3" * SIN(3 * 0.4 * "x") + "w0d_6_6_3" * COS(3 * 0.4 * "x");
    "phi" := "phi" + "w0c_6_6_4" * SIN(4 * 0.4 * "x") + "w0d_6_6_4" * COS(4 * 0.4 * "x");
    "phi" := "phi" + "w0c_6_6_5" * SIN(5 * 0.4 * "x") + "w0d_6_6_5" * COS(5 * 0.4 * "x");
    "phi" := "phi" + "w0c_6_6_6" * SIN(6 * 0.4 * "x") + "w0d_6_6_6" * COS(6 * 0.4 * "x");
    "acc" := "acc" + "phi";
    "x" := "feat_7";
    "phi" := "w0b_6_7" * "x" / (1.0 + EXP(-"x"));
    "phi" := "phi" + "w0c_6_7_1" * SIN(1 * 0.4 * "x") + "w0d_6_7_1" * COS(1 * 0.4 * "x");
    "phi" := "phi" + "w0c_6_7_2" * SIN(2 * 0.4 * "x") + "w0d_6_7_2" * COS(2 * 0.4 * "x");
    "phi" := "phi" + "w0c_6_7_3" * SIN(3 * 0.4 * "x") + "w0d_6_7_3" * COS(3 * 0.4 * "x");
    "phi" := "phi" + "w0c_6_7_4" * SIN(4 * 0.4 * "x") + "w0d_6_7_4" * COS(4 * 0.4 * "x");
    "phi" := "phi" + "w0c_6_7_5" * SIN(5 * 0.4 * "x") + "w0d_6_7_5" * COS(5 * 0.4 * "x");
    "phi" := "phi" + "w0c_6_7_6" * SIN(6 * 0.4 * "x") + "w0d_6_7_6" * COS(6 * 0.4 * "x");
    "acc" := "acc" + "phi";
    "x" := "feat_8";
    "phi" := "w0b_6_8" * "x" / (1.0 + EXP(-"x"));
    "phi" := "phi" + "w0c_6_8_1" * SIN(1 * 0.4 * "x") + "w0d_6_8_1" * COS(1 * 0.4 * "x");
    "phi" := "phi" + "w0c_6_8_2" * SIN(2 * 0.4 * "x") + "w0d_6_8_2" * COS(2 * 0.4 * "x");
    "phi" := "phi" + "w0c_6_8_3" * SIN(3 * 0.4 * "x") + "w0d_6_8_3" * COS(3 * 0.4 * "x");
    "phi" := "phi" + "w0c_6_8_4" * SIN(4 * 0.4 * "x") + "w0d_6_8_4" * COS(4 * 0.4 * "x");
    "phi" := "phi" + "w0c_6_8_5" * SIN(5 * 0.4 * "x") + "w0d_6_8_5" * COS(5 * 0.4 * "x");
    "phi" := "phi" + "w0c_6_8_6" * SIN(6 * 0.4 * "x") + "w0d_6_8_6" * COS(6 * 0.4 * "x");
    "acc" := "acc" + "phi";
    "x" := "feat_9";
    "phi" := "w0b_6_9" * "x" / (1.0 + EXP(-"x"));
    "phi" := "phi" + "w0c_6_9_1" * SIN(1 * 0.4 * "x") + "w0d_6_9_1" * COS(1 * 0.4 * "x");
    "phi" := "phi" + "w0c_6_9_2" * SIN(2 * 0.4 * "x") + "w0d_6_9_2" * COS(2 * 0.4 * "x");
    "phi" := "phi" + "w0c_6_9_3" * SIN(3 * 0.4 * "x") + "w0d_6_9_3" * COS(3 * 0.4 * "x");
    "phi" := "phi" + "w0c_6_9_4" * SIN(4 * 0.4 * "x") + "w0d_6_9_4" * COS(4 * 0.4 * "x");
    "phi" := "phi" + "w0c_6_9_5" * SIN(5 * 0.4 * "x") + "w0d_6_9_5" * COS(5 * 0.4 * "x");
    "phi" := "phi" + "w0c_6_9_6" * SIN(6 * 0.4 * "x") + "w0d_6_9_6" * COS(6 * 0.4 * "x");
    "acc" := "acc" + "phi";
    "x" := "feat_10";
    "phi" := "w0b_6_10" * "x" / (1.0 + EXP(-"x"));
    "phi" := "phi" + "w0c_6_10_1" * SIN(1 * 0.4 * "x") + "w0d_6_10_1" * COS(1 * 0.4 * "x");
    "phi" := "phi" + "w0c_6_10_2" * SIN(2 * 0.4 * "x") + "w0d_6_10_2" * COS(2 * 0.4 * "x");
    "phi" := "phi" + "w0c_6_10_3" * SIN(3 * 0.4 * "x") + "w0d_6_10_3" * COS(3 * 0.4 * "x");
    "phi" := "phi" + "w0c_6_10_4" * SIN(4 * 0.4 * "x") + "w0d_6_10_4" * COS(4 * 0.4 * "x");
    "phi" := "phi" + "w0c_6_10_5" * SIN(5 * 0.4 * "x") + "w0d_6_10_5" * COS(5 * 0.4 * "x");
    "phi" := "phi" + "w0c_6_10_6" * SIN(6 * 0.4 * "x") + "w0d_6_10_6" * COS(6 * 0.4 * "x");
    "acc" := "acc" + "phi";
    "x" := "feat_11";
    "phi" := "w0b_6_11" * "x" / (1.0 + EXP(-"x"));
    "phi" := "phi" + "w0c_6_11_1" * SIN(1 * 0.4 * "x") + "w0d_6_11_1" * COS(1 * 0.4 * "x");
    "phi" := "phi" + "w0c_6_11_2" * SIN(2 * 0.4 * "x") + "w0d_6_11_2" * COS(2 * 0.4 * "x");
    "phi" := "phi" + "w0c_6_11_3" * SIN(3 * 0.4 * "x") + "w0d_6_11_3" * COS(3 * 0.4 * "x");
    "phi" := "phi" + "w0c_6_11_4" * SIN(4 * 0.4 * "x") + "w0d_6_11_4" * COS(4 * 0.4 * "x");
    "phi" := "phi" + "w0c_6_11_5" * SIN(5 * 0.4 * "x") + "w0d_6_11_5" * COS(5 * 0.4 * "x");
    "phi" := "phi" + "w0c_6_11_6" * SIN(6 * 0.4 * "x") + "w0d_6_11_6" * COS(6 * 0.4 * "x");
    "acc" := "acc" + "phi";
    "x" := "feat_12";
    "phi" := "w0b_6_12" * "x" / (1.0 + EXP(-"x"));
